// TIA Portal V17 export
// export: Created 2023-02-14T02:49:17.7051188Z, ExportSetting WithDefaults, DisplayName Totally Integrated Automation Portal, DisplayVersion V17, DisplayName TIA Portal Openness, DisplayVersion V17, DisplayName TIA Portal Teamcenter Gateway, DisplayVersion V17, DisplayName TIA Portal Version Control Interface, DisplayVersion V17, DisplayName SINAMICS Startdrive Advanced, DisplayVersion V17, DisplayName SINAMICS Startdrive G130, G150, S120, S150, SINAMICS MV, S210, DisplayVersion V17, DisplayName SINAMICS Startdrive G110M, G120, G120C, G120D, G120P, G115D, DisplayVersion V17, DisplayName STEP 7 Professional, DisplayVersion V17, DisplayName STEP 7 Safety, DisplayVersion V17, DisplayName WinCC Professional, DisplayVersion V17
FUNCTION "BlendingArea" : Void   // FC201, LAD
{ S7_Optimized_Access := 'TRUE' }
VERSION : 0.1
// stored: AutoNumber false, IsIECCheckEnabled false, SetENOAutomatically false, UDAEnableTagReadback false
   VAR_TEMP   // added for the SCL form of the ladder/FBD networks
      _w1 : Bool;
      _w2 : Bool;
   END_VAR
BEGIN

REGION Network 1: Analog
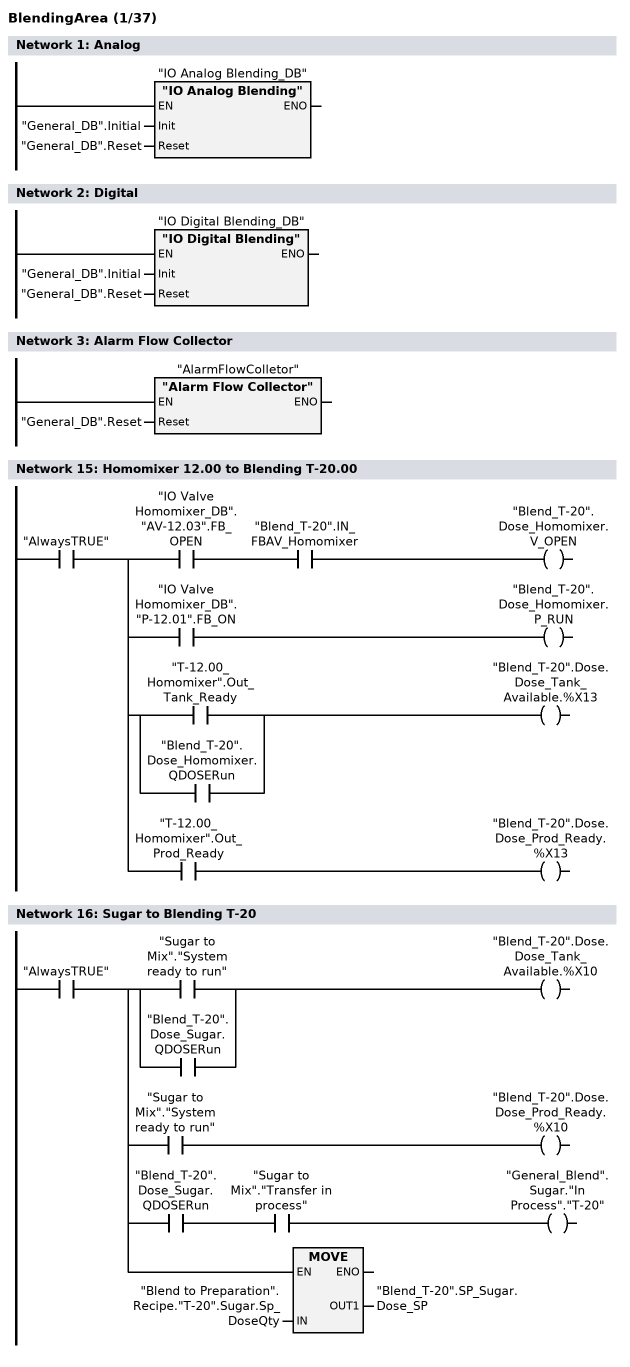
   RUNG wire#powerrail
      "IO Analog Blending_DB"(Init := "General_DB".Initial, Reset := "General_DB".Reset)
   END_RUNG
   // the same network as SCL:
   "IO Analog Blending_DB"(Init := "General_DB".Initial, Reset := "General_DB".Reset);   // "IO Analog Blending"
END_REGION

REGION Network 2: Digital
   RUNG wire#powerrail
      "IO Digital Blending_DB"(Init := "General_DB".Initial, Reset := "General_DB".Reset)
   END_RUNG
   // the same network as SCL:
   "IO Digital Blending_DB"(Init := "General_DB".Initial, Reset := "General_DB".Reset);   // "IO Digital Blending"
END_REGION

REGION Network 3: Alarm Flow Collector
   RUNG wire#powerrail
      "AlarmFlowColletor"(Reset := "General_DB".Reset)
   END_RUNG
   // the same network as SCL:
   "AlarmFlowColletor"(Reset := "General_DB".Reset);   // "Alarm Flow Collector"
END_REGION

NETWORK
TITLE = ChiliAwetan1 to Blending T-20
//Valve Open
      A     "Preparation to Blend"."T-02_ChiliAwetan_1".Valve_Open;
      A(;
      O(;
      A     "Blend_T-20".Dose.Dose_Header_Req.%X0;
      A     "Blend_T-20".IN_FBAV_Header1;
      );
      O(;
      A     "Blend_T-20".Dose.Dose_Header_Req.%X16;
      A     "Blend_T-20".IN_FBAV_Header2;
      );
      );
      =     "Blend_T-20".Dose_ChiliAwetan1.V_OPEN;
//Pump On
      O     "Preparation to Blend"."T-02_ChiliAwetan_1".Pump_Run;
      =     "Blend_T-20".Dose_ChiliAwetan1.P_RUN;
//Tank Available
      O     "Preparation to Blend"."T-02_ChiliAwetan_1".Tank_Available;
      O     "Blend_T-20".Dose_ChiliAwetan1.QDOSERun;
      =     "Blend_T-20".Dose.Dose_Tank_Available.%X0;
//Product Ready
      O     "Preparation to Blend"."T-02_ChiliAwetan_1".Product_Ready;
      =     "Blend_T-20".Dose.Dose_Prod_Ready.%X0;
//Level Tank
      L     "Preparation to Blend"."T-02_ChiliAwetan_1".Level;
      T     "Blend_T-20"."Dose_Level_%"."ChiliAwetan1%";


NETWORK
TITLE = ChiliAwetan2 to Blending T-20
//Valve Open
      A     "Preparation to Blend"."T-03_ChiliAwetan_2".Valve_Open;
      A(;
      O(;
      A     "Blend_T-20".Dose.Dose_Header_Req.%X1;
      A     "Blend_T-20".IN_FBAV_Header1;
      );
      O(;
      A     "Blend_T-20".Dose.Dose_Header_Req.%X17;
      A     "Blend_T-20".IN_FBAV_Header2;
      );
      );
      =     "Blend_T-20".Dose_ChiliAwetan2.V_OPEN;
//Pump On
      O     "Preparation to Blend"."T-03_ChiliAwetan_2".Pump_Run;
      =     "Blend_T-20".Dose_ChiliAwetan2.P_RUN;
//Tank Available
      O     "Preparation to Blend"."T-03_ChiliAwetan_2".Tank_Available;
      O     "Blend_T-20".Dose_ChiliAwetan2.QDOSERun;
      =     "Blend_T-20".Dose.Dose_Tank_Available.%X1;
//Product Ready
      O     "Preparation to Blend"."T-03_ChiliAwetan_2".Product_Ready;
      =     "Blend_T-20".Dose.Dose_Prod_Ready.%X1;
//Level Tank
      L     "Preparation to Blend"."T-03_ChiliAwetan_2".Level;
      T     "Blend_T-20"."Dose_Level_%"."ChiliAwetan2%";


NETWORK
TITLE = ChiliAwetan3 to Blending T-20
//Valve Open
      A     "Preparation to Blend"."T-04_ChiliAwetan_3".Valve_Open;
      A(;
      O(;
      A     "Blend_T-20".Dose.Dose_Header_Req.%X2;
      A     "Blend_T-20".IN_FBAV_Header1;
      );
      O(;
      A     "Blend_T-20".Dose.Dose_Header_Req.%X18;
      A     "Blend_T-20".IN_FBAV_Header2;
      );
      );
      =     "Blend_T-20".Dose_ChiliAwetan3.V_OPEN;
//Pump On
      O     "Preparation to Blend"."T-04_ChiliAwetan_3".Pump_Run;
      =     "Blend_T-20".Dose_ChiliAwetan3.P_RUN;
//Tank Available
      O     "Preparation to Blend"."T-04_ChiliAwetan_3".Tank_Available;
      O     "Blend_T-20".Dose_ChiliAwetan3.QDOSERun;
      =     "Blend_T-20".Dose.Dose_Tank_Available.%X2;
//Product Ready
      O     "Preparation to Blend"."T-04_ChiliAwetan_3".Product_Ready;
      =     "Blend_T-20".Dose.Dose_Prod_Ready.%X2;
//Level Tank
      L     "Preparation to Blend"."T-04_ChiliAwetan_3".Level;
      T     "Blend_T-20"."Dose_Level_%"."ChiliAwetan3%";


NETWORK
TITLE = Tomato to Blending T-20
//Valve Open
      A     "Preparation to Blend"."T-05_Tomato".Valve_Open;
      A(;
      O(;
      A     "Blend_T-20".Dose.Dose_Header_Req.%X3;
      A     "Blend_T-20".IN_FBAV_Header1;
      );
      O(;
      A     "Blend_T-20".Dose.Dose_Header_Req.%X19;
      A     "Blend_T-20".IN_FBAV_Header2;
      );
      );
      =     "Blend_T-20".Dose_Tomato.V_OPEN;
//Pump On
      O     "Preparation to Blend"."T-05_Tomato".Pump_Run;
      =     "Blend_T-20".Dose_Tomato.P_RUN;
//Tank Available
      O     "Preparation to Blend"."T-05_Tomato".Tank_Available;
      O     "Blend_T-20".Dose_Tomato.QDOSERun;
      =     "Blend_T-20".Dose.Dose_Tank_Available.%X3;
//Product Ready
      O     "Preparation to Blend"."T-05_Tomato".Product_Ready;
      =     "Blend_T-20".Dose.Dose_Prod_Ready.%X3;
//Level Tank
      L     "Preparation to Blend"."T-05_Tomato".Level;
      T     "Blend_T-20"."Dose_Level_%"."Tomato%";


NETWORK
TITLE = ChiliFresh1 to Blending T-20
//Valve Open
      A     "Preparation to Blend"."T-06_ChiliFresh_1".Valve_Open;
      A(;
      O(;
      A     "Blend_T-20".Dose.Dose_Header_Req.%X4;
      A     "Blend_T-20".IN_FBAV_Header1;
      );
      O(;
      A     "Blend_T-20".Dose.Dose_Header_Req.%X20;
      A     "Blend_T-20".IN_FBAV_Header2;
      );
      );
      =     "Blend_T-20".Dose_ChiliFresh1.V_OPEN;
//Pump On
      O     "Preparation to Blend"."T-06_ChiliFresh_1".Pump_Run;
      =     "Blend_T-20".Dose_ChiliFresh1.P_RUN;
//Tank Available
      O     "Preparation to Blend"."T-06_ChiliFresh_1".Tank_Available;
      O     "Blend_T-20".Dose_ChiliFresh1.QDOSERun;
      =     "Blend_T-20".Dose.Dose_Tank_Available.%X4;
//Product Ready
      O     "Preparation to Blend"."T-06_ChiliFresh_1".Product_Ready;
      =     "Blend_T-20".Dose.Dose_Prod_Ready.%X4;
//Level Tank
      L     "Preparation to Blend"."T-06_ChiliFresh_1".Level;
      T     "Blend_T-20"."Dose_Level_%"."ChiliFresh1%";


NETWORK
TITLE = ChiliFresh2 to Blending T-20
//Valve Open
      A     "Preparation to Blend"."T-07_ChiliFresh_2".Valve_Open;
      A(;
      O(;
      A     "Blend_T-20".Dose.Dose_Header_Req.%X5;
      A     "Blend_T-20".IN_FBAV_Header1;
      );
      O(;
      A     "Blend_T-20".Dose.Dose_Header_Req.%X21;
      A     "Blend_T-20".IN_FBAV_Header2;
      );
      );
      =     "Blend_T-20".Dose_ChiliFresh2.V_OPEN;
//Pump On
      O     "Preparation to Blend"."T-07_ChiliFresh_2".Pump_Run;
      =     "Blend_T-20".Dose_ChiliFresh2.P_RUN;
//Tank Available
      O     "Preparation to Blend"."T-07_ChiliFresh_2".Tank_Available;
      O     "Blend_T-20".Dose_ChiliFresh2.QDOSERun;
      =     "Blend_T-20".Dose.Dose_Tank_Available.%X5;
//Product Ready
      O     "Preparation to Blend"."T-07_ChiliFresh_2".Product_Ready;
      =     "Blend_T-20".Dose.Dose_Prod_Ready.%X5;
//Level Tank
      L     "Preparation to Blend"."T-07_ChiliFresh_2".Level;
      T     "Blend_T-20"."Dose_Level_%"."ChiliFresh2%";


NETWORK
TITLE = ChiliFresh3 to Blending T-20
//Valve Open
      A     "Preparation to Blend"."T-08_ChiliFresh_3".Valve_Open;
      A(;
      O(;
      A     "Blend_T-20".Dose.Dose_Header_Req.%X6;
      A     "Blend_T-20".IN_FBAV_Header1;
      );
      O(;
      A     "Blend_T-20".Dose.Dose_Header_Req.%X22;
      A     "Blend_T-20".IN_FBAV_Header2;
      );
      );
      =     "Blend_T-20".Dose_ChiliFresh3.V_OPEN;
//Pump On
      O     "Preparation to Blend"."T-08_ChiliFresh_3".Pump_Run;
      =     "Blend_T-20".Dose_ChiliFresh3.P_RUN;
//Tank Available
      O     "Preparation to Blend"."T-08_ChiliFresh_3".Tank_Available;
      O     "Blend_T-20".Dose_ChiliFresh3.QDOSERun;
      =     "Blend_T-20".Dose.Dose_Tank_Available.%X6;
//Product Ready
      O     "Preparation to Blend"."T-08_ChiliFresh_3".Product_Ready;
      =     "Blend_T-20".Dose.Dose_Prod_Ready.%X6;
//Level Tank
      L     "Preparation to Blend"."T-08_ChiliFresh_3".Level;
      T     "Blend_T-20"."Dose_Level_%"."ChiliFresh3%";


NETWORK
TITLE = Garlic to Blending T-20
//Valve Open
      A     "Preparation to Blend"."T-09_Garlic".Valve_Open;
      A(;
      O(;
      A     "Blend_T-20".Dose.Dose_Header_Req.%X7;
      A     "Blend_T-20".IN_FBAV_Header1;
      );
      O(;
      A     "Blend_T-20".Dose.Dose_Header_Req.%X23;
      A     "Blend_T-20".IN_FBAV_Header2;
      );
      );
      =     "Blend_T-20".Dose_Garlic.V_OPEN;
//Pump On
      O     "Preparation to Blend"."T-09_Garlic".Pump_Run;
      =     "Blend_T-20".Dose_Garlic.P_RUN;
//Tank Available
      O     "Preparation to Blend"."T-09_Garlic".Tank_Available;
      O     "Blend_T-20".Dose_Garlic.QDOSERun;
      =     "Blend_T-20".Dose.Dose_Tank_Available.%X7;
//Product Ready
      O     "Preparation to Blend"."T-09_Garlic".Product_Ready;
      =     "Blend_T-20".Dose.Dose_Prod_Ready.%X7;
//Level Tank
      L     "Preparation to Blend"."T-09_Garlic".Level;
      T     "Blend_T-20"."Dose_Level_%"."Garlic%";


NETWORK
TITLE = Vinegar to Blending T-20
//Valve Open
      A     "Preparation to Blend"."T-10_Vinegar".Valve_Open;
      A     "Blend_T-20".IN_FBAV_Vinegar;
      =     "Blend_T-20".Dose_Vinegar.V_OPEN;
//Pump On
      O     "Preparation to Blend"."T-10_Vinegar".Pump_Run;
      =     "Blend_T-20".Dose_Vinegar.P_RUN;
//Tank Available
      O     "Preparation to Blend"."T-10_Vinegar".Tank_Available;
      O     "Blend_T-20".Dose_Vinegar.QDOSERun;
      =     "Blend_T-20".Dose.Dose_Tank_Available.%X9;
//Product Ready
      O     "Preparation to Blend"."T-10_Vinegar".Product_Ready;
      =     "Blend_T-20".Dose.Dose_Prod_Ready.%X9;
//Level Tank
      L     "Preparation to Blend"."T-10_Vinegar".Level;
      T     "Blend_T-20"."Dose_Level_%"."Vinegar%";


NETWORK
TITLE = HW to Blending T-20
//Valve Open
      A     "Preparation to Blend"."T-51_HW".Valve_Open;
      A(;
      O(;
      A     "Blend_T-20".Dose.Dose_Header_Req.%X8;
      A     "Blend_T-20".IN_FBAV_Header1;
      );
      O(;
      A     "Blend_T-20".Dose.Dose_Header_Req.%X24;
      A     "Blend_T-20".IN_FBAV_Header2;
      );
      );
      =     "Blend_T-20".Dose_HW.V_OPEN;
//Pump On
      O     "Preparation to Blend"."T-51_HW".Pump_Run;
      =     "Blend_T-20".Dose_HW.P_RUN;
//Tank Available
      O     "Preparation to Blend"."T-51_HW".Tank_Available;
      O     "Blend_T-20".Dose_HW.QDOSERun;
      =     "Blend_T-20".Dose.Dose_Tank_Available.%X8;
//Product Ready
      O     "Preparation to Blend"."T-51_HW".Product_Ready;
      =     "Blend_T-20".Dose.Dose_Prod_Ready.%X8;
//Level Tank
// L     "Preparation to Blend"."T-01_HW".Level
// T     "Blend_T-20"."Dose_Level_%"."HW%"


REGION Network 15: Homomixer 12.00 to Blending T-20.00
   RUNG wire#powerrail
      Contact( "AlwaysTRUE" )
      wire#w1
      Contact( "IO Valve Homomixer_DB"."AV-12.03".FB_OPEN )
      Contact( "Blend_T-20".IN_FBAV_Homomixer )
      Coil( "Blend_T-20".Dose_Homomixer.V_OPEN )
   END_RUNG
   RUNG wire#w1
      Contact( "IO Valve Homomixer_DB"."P-12.01".FB_ON )
      Coil( "Blend_T-20".Dose_Homomixer.P_RUN )
   END_RUNG
   RUNG wire#w1
      Contact( "T-12.00_Homomixer".Out_Tank_Ready )
      wire#w2
      Coil( "Blend_T-20".Dose.Dose_Tank_Available.%X13 )
   END_RUNG
   RUNG wire#w1
      Contact( "Blend_T-20".Dose_Homomixer.QDOSERun )
   END_RUNG wire#w2
   RUNG wire#w1
      Contact( "T-12.00_Homomixer".Out_Prod_Ready )
      Coil( "Blend_T-20".Dose.Dose_Prod_Ready.%X13 )
   END_RUNG
   // the same network as SCL:
   "Blend_T-20".Dose_Homomixer.V_OPEN := "AlwaysTRUE" AND "IO Valve Homomixer_DB"."AV-12.03".FB_OPEN AND "Blend_T-20".IN_FBAV_Homomixer;
   "Blend_T-20".Dose_Homomixer.P_RUN := "AlwaysTRUE" AND "IO Valve Homomixer_DB"."P-12.01".FB_ON;
   "Blend_T-20".Dose.Dose_Tank_Available.%X13 := "AlwaysTRUE" AND ("T-12.00_Homomixer".Out_Tank_Ready OR "Blend_T-20".Dose_Homomixer.QDOSERun);
   "Blend_T-20".Dose.Dose_Prod_Ready.%X13 := "AlwaysTRUE" AND "T-12.00_Homomixer".Out_Prod_Ready;
END_REGION

REGION Network 16: Sugar to Blending T-20
   RUNG wire#powerrail
      Contact( "AlwaysTRUE" )
      wire#w1
      Contact( "Sugar to Mix"."System ready to run" )
      wire#w2
      Coil( "Blend_T-20".Dose.Dose_Tank_Available.%X10 )
   END_RUNG
   RUNG wire#w1
      Contact( "Blend_T-20".Dose_Sugar.QDOSERun )
   END_RUNG wire#w2
   RUNG wire#w1
      Contact( "Sugar to Mix"."System ready to run" )
      Coil( "Blend_T-20".Dose.Dose_Prod_Ready.%X10 )
   END_RUNG
   RUNG wire#w1
      Contact( "Blend_T-20".Dose_Sugar.QDOSERun )
      Contact( "Sugar to Mix"."Transfer in process" )
      Coil( "General_Blend".Sugar."In Process"."T-20" )
   END_RUNG
   RUNG wire#w1
      Move(in := "Blend to Preparation".Recipe."T-20".Sugar.Sp_DoseQty, out1 => "Blend_T-20".SP_Sugar.Dose_SP)
   END_RUNG
   // the same network as SCL:
   "Blend_T-20".Dose.Dose_Tank_Available.%X10 := "AlwaysTRUE" AND ("Sugar to Mix"."System ready to run" OR "Blend_T-20".Dose_Sugar.QDOSERun);
   "Blend_T-20".Dose.Dose_Prod_Ready.%X10 := "AlwaysTRUE" AND "Sugar to Mix"."System ready to run";
   "General_Blend".Sugar."In Process"."T-20" := "AlwaysTRUE" AND "Blend_T-20".Dose_Sugar.QDOSERun AND "Sugar to Mix"."Transfer in process";
   IF "AlwaysTRUE" THEN
       "Blend_T-20".SP_Sugar.Dose_SP := "Blend to Preparation".Recipe."T-20".Sugar.Sp_DoseQty;
   END_IF;
END_REGION

REGION Network 17: Salt to Blending T-20
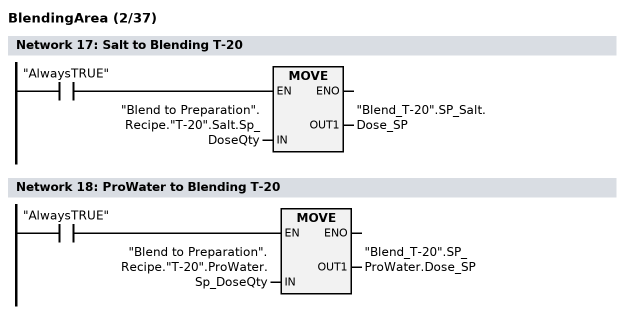
   RUNG wire#powerrail
      Contact( "AlwaysTRUE" )
      Move(in := "Blend to Preparation".Recipe."T-20".Salt.Sp_DoseQty, out1 => "Blend_T-20".SP_Salt.Dose_SP)
   END_RUNG
   // the same network as SCL:
   IF "AlwaysTRUE" THEN
       "Blend_T-20".SP_Salt.Dose_SP := "Blend to Preparation".Recipe."T-20".Salt.Sp_DoseQty;
   END_IF;
END_REGION

REGION Network 18: ProWater to Blending T-20
   RUNG wire#powerrail
      Contact( "AlwaysTRUE" )
      Move(in := "Blend to Preparation".Recipe."T-20".ProWater.Sp_DoseQty, out1 => "Blend_T-20".SP_ProWater.Dose_SP)
   END_RUNG
   // the same network as SCL:
   IF "AlwaysTRUE" THEN
       "Blend_T-20".SP_ProWater.Dose_SP := "Blend to Preparation".Recipe."T-20".ProWater.Sp_DoseQty;
   END_IF;
END_REGION

REGION Network 19: Blending T-20
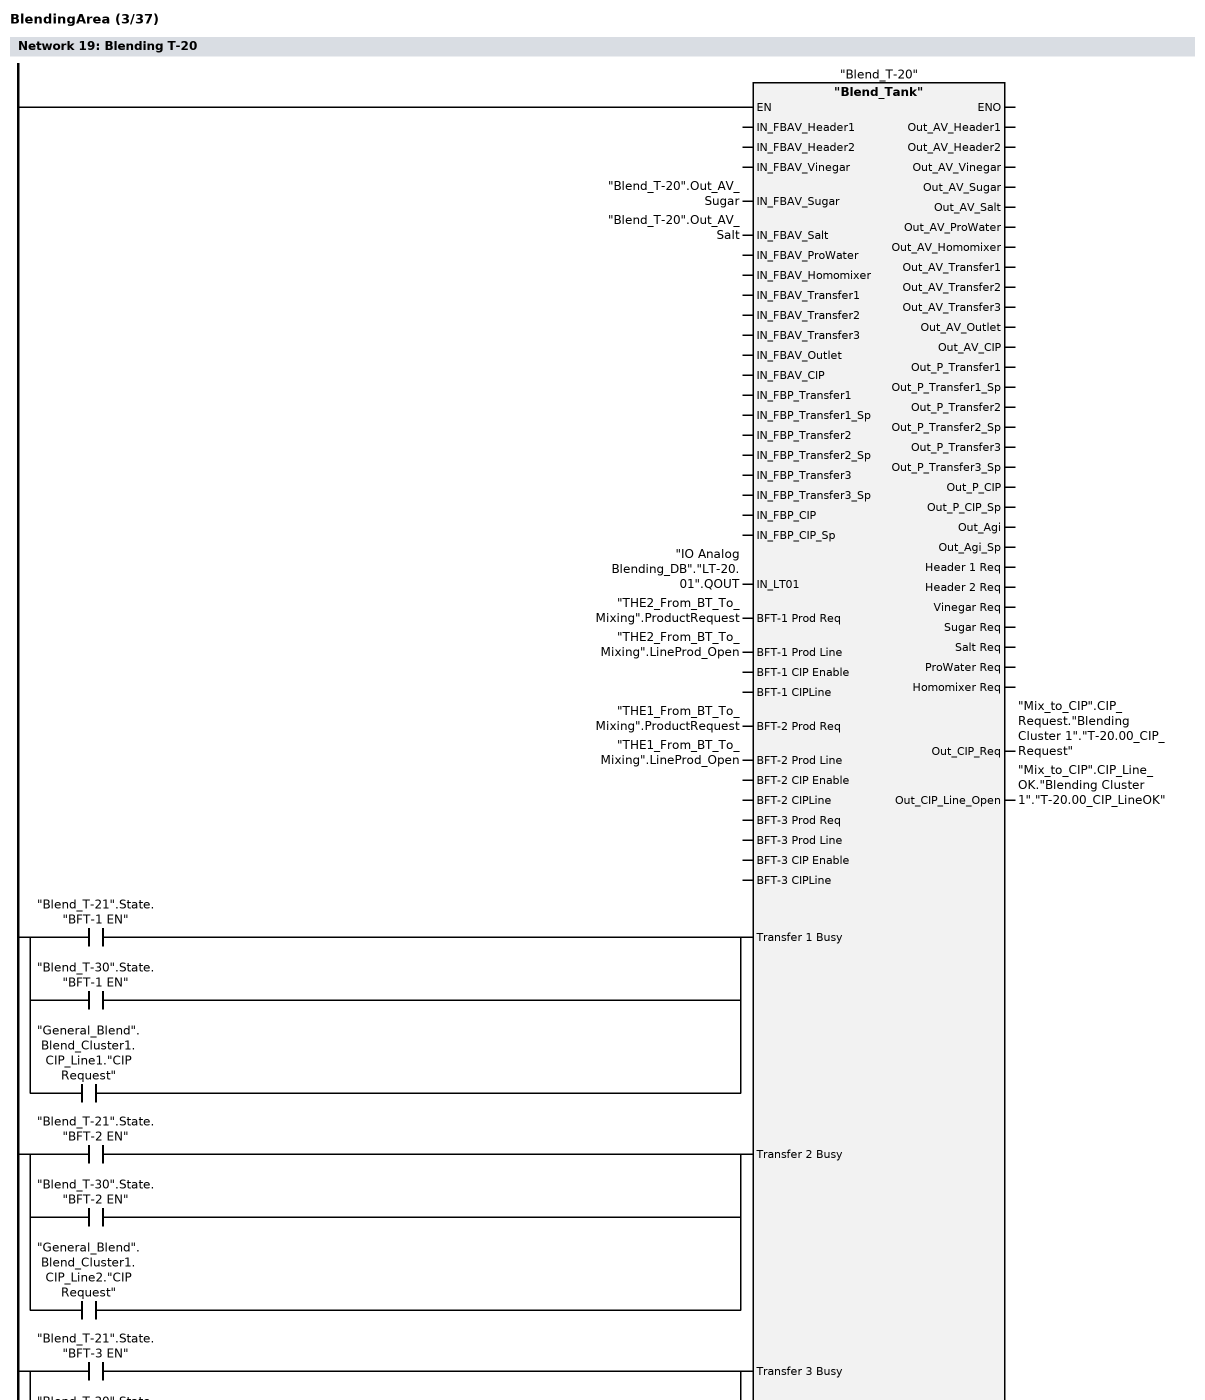
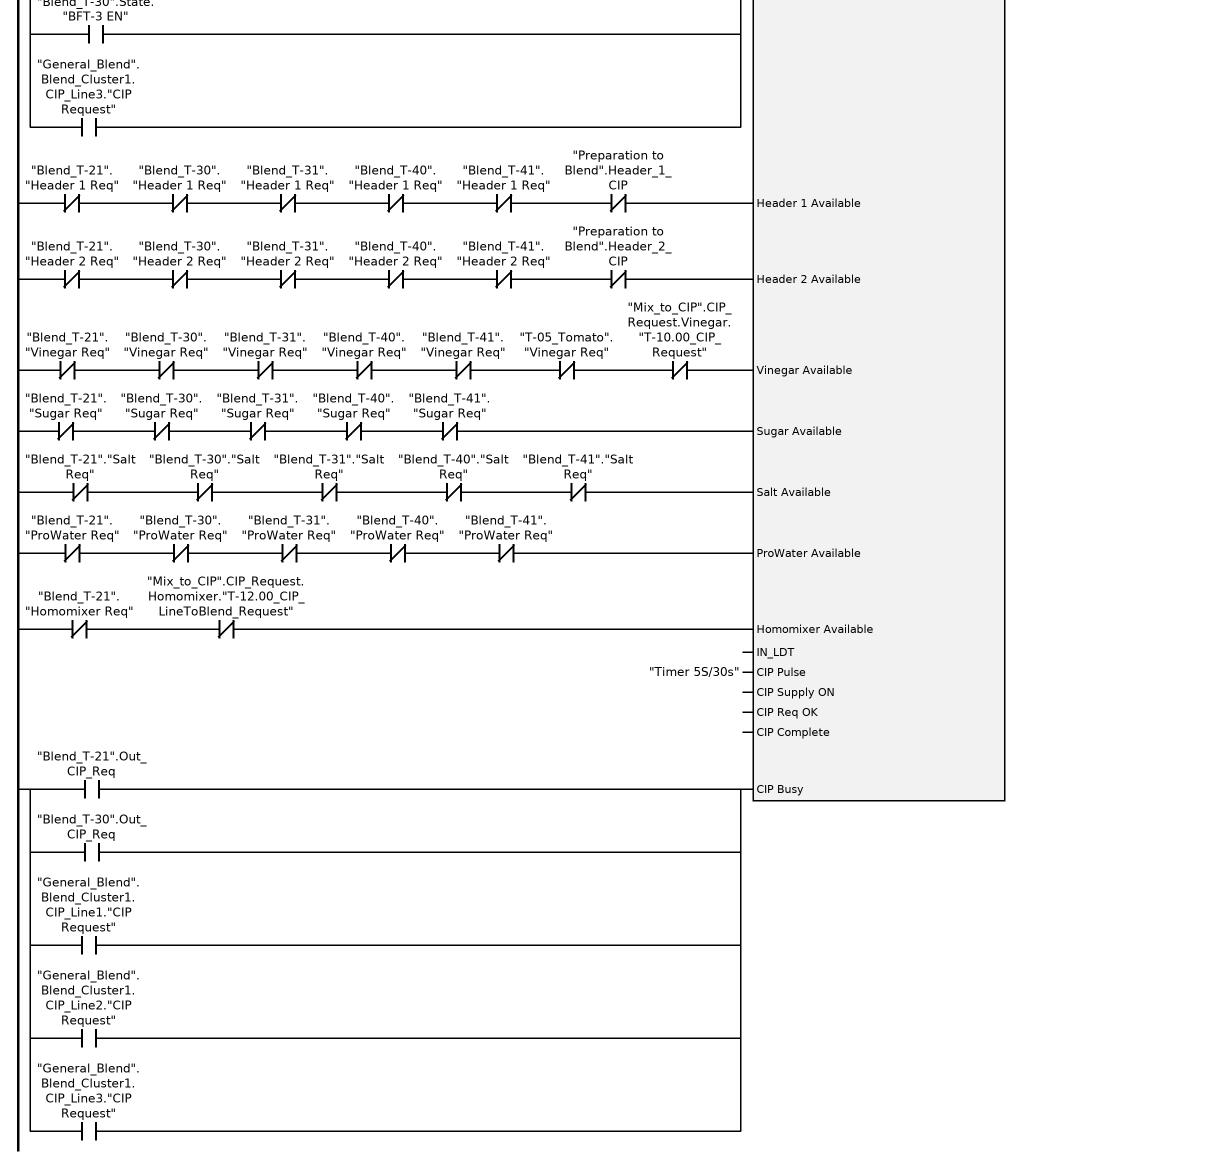
   RUNG wire#powerrail
      "Blend_T-20"("Transfer 1 Busy" := wire#w1, "Transfer 2 Busy" := wire#w2, "Transfer 3 Busy" := wire#w3, "Header 1 Available" := wire#w4, "Header 2 Available" := wire#w5, "Vinegar Available" := wire#w6, "Sugar Available" := wire#w7, "Salt Available" := wire#w8, "ProWater Available" := wire#w9, "Homomixer Available" := wire#w10, "CIP Busy" := wire#w11, IN_FBAV_Header1 :=, IN_FBAV_Header2 :=, IN_FBAV_Vinegar :=, IN_FBAV_Sugar := "Blend_T-20".Out_AV_Sugar, IN_FBAV_Salt := "Blend_T-20".Out_AV_Salt, IN_FBAV_ProWater :=, IN_FBAV_Homomixer :=, IN_FBAV_Transfer1 :=, IN_FBAV_Transfer2 :=, IN_FBAV_Transfer3 :=, IN_FBAV_Outlet :=, IN_FBAV_CIP :=, IN_FBP_Transfer1 :=, IN_FBP_Transfer1_Sp :=, IN_FBP_Transfer2 :=, IN_FBP_Transfer2_Sp :=, IN_FBP_Transfer3 :=, IN_FBP_Transfer3_Sp :=, IN_FBP_CIP :=, IN_FBP_CIP_Sp :=, IN_LT01 := "IO Analog Blending_DB"."LT-20.01".QOUT, "BFT-1 Prod Req" := "THE2_From_BT_To_Mixing".ProductRequest, "BFT-1 Prod Line" := "THE2_From_BT_To_Mixing".LineProd_Open, "BFT-1 CIP Enable" :=, "BFT-1 CIPLine" :=, "BFT-2 Prod Req" := "THE1_From_BT_To_Mixing".ProductRequest, "BFT-2 Prod Line" := "THE1_From_BT_To_Mixing".LineProd_Open, "BFT-2 CIP Enable" :=, "BFT-2 CIPLine" :=, "BFT-3 Prod Req" :=, "BFT-3 Prod Line" :=, "BFT-3 CIP Enable" :=, "BFT-3 CIPLine" :=, IN_LDT :=, "CIP Pulse" := "Timer 5S/30s", "CIP Supply ON" :=, "CIP Req OK" :=, "CIP Complete" :=, Out_AV_Header1 =>, Out_AV_Header2 =>, Out_AV_Vinegar =>, Out_AV_Sugar =>, Out_AV_Salt =>, Out_AV_ProWater =>, Out_AV_Homomixer =>, Out_AV_Transfer1 =>, Out_AV_Transfer2 =>, Out_AV_Transfer3 =>, Out_AV_Outlet =>, Out_AV_CIP =>, Out_P_Transfer1 =>, Out_P_Transfer1_Sp =>, Out_P_Transfer2 =>, Out_P_Transfer2_Sp =>, Out_P_Transfer3 =>, Out_P_Transfer3_Sp =>, Out_P_CIP =>, Out_P_CIP_Sp =>, Out_Agi =>, Out_Agi_Sp =>, "Header 1 Req" =>, "Header 2 Req" =>, "Vinegar Req" =>, "Sugar Req" =>, "Salt Req" =>, "ProWater Req" =>, "Homomixer Req" =>, Out_CIP_Req => "Mix_to_CIP".CIP_Request."Blending Cluster 1"."T-20.00_CIP_Request", Out_CIP_Line_Open => "Mix_to_CIP".CIP_Line_OK."Blending Cluster 1"."T-20.00_CIP_LineOK")
   END_RUNG
   RUNG wire#powerrail
      Contact( "Blend_T-21".State."BFT-1 EN" )
   END_RUNG wire#w1
   RUNG wire#powerrail
      Contact( "Blend_T-30".State."BFT-1 EN" )
   END_RUNG wire#w1
   RUNG wire#powerrail
      Contact( "General_Blend".Blend_Cluster1.CIP_Line1."CIP Request" )
   END_RUNG wire#w1
   RUNG wire#powerrail
      Contact( "Blend_T-21".State."BFT-2 EN" )
   END_RUNG wire#w2
   RUNG wire#powerrail
      Contact( "Blend_T-30".State."BFT-2 EN" )
   END_RUNG wire#w2
   RUNG wire#powerrail
      Contact( "General_Blend".Blend_Cluster1.CIP_Line2."CIP Request" )
   END_RUNG wire#w2
   RUNG wire#powerrail
      Contact( "Blend_T-21".State."BFT-3 EN" )
   END_RUNG wire#w3
   RUNG wire#powerrail
      Contact( "Blend_T-30".State."BFT-3 EN" )
   END_RUNG wire#w3
   RUNG wire#powerrail
      Contact( "General_Blend".Blend_Cluster1.CIP_Line3."CIP Request" )
   END_RUNG wire#w3
   RUNG wire#powerrail
      I_Contact( "Blend_T-21"."Header 1 Req" )
      I_Contact( "Blend_T-30"."Header 1 Req" )
      I_Contact( "Blend_T-31"."Header 1 Req" )
      I_Contact( "Blend_T-40"."Header 1 Req" )
      I_Contact( "Blend_T-41"."Header 1 Req" )
      I_Contact( "Preparation to Blend".Header_1_CIP )
   END_RUNG wire#w4
   RUNG wire#powerrail
      I_Contact( "Blend_T-21"."Header 2 Req" )
      I_Contact( "Blend_T-30"."Header 2 Req" )
      I_Contact( "Blend_T-31"."Header 2 Req" )
      I_Contact( "Blend_T-40"."Header 2 Req" )
      I_Contact( "Blend_T-41"."Header 2 Req" )
      I_Contact( "Preparation to Blend".Header_2_CIP )
   END_RUNG wire#w5
   RUNG wire#powerrail
      I_Contact( "Blend_T-21"."Vinegar Req" )
      I_Contact( "Blend_T-30"."Vinegar Req" )
      I_Contact( "Blend_T-31"."Vinegar Req" )
      I_Contact( "Blend_T-40"."Vinegar Req" )
      I_Contact( "Blend_T-41"."Vinegar Req" )
      I_Contact( "T-05_Tomato"."Vinegar Req" )
      I_Contact( "Mix_to_CIP".CIP_Request.Vinegar."T-10.00_CIP_Request" )
   END_RUNG wire#w6
   RUNG wire#powerrail
      I_Contact( "Blend_T-21"."Sugar Req" )
      I_Contact( "Blend_T-30"."Sugar Req" )
      I_Contact( "Blend_T-31"."Sugar Req" )
      I_Contact( "Blend_T-40"."Sugar Req" )
      I_Contact( "Blend_T-41"."Sugar Req" )
   END_RUNG wire#w7
   RUNG wire#powerrail
      I_Contact( "Blend_T-21"."Salt Req" )
      I_Contact( "Blend_T-30"."Salt Req" )
      I_Contact( "Blend_T-31"."Salt Req" )
      I_Contact( "Blend_T-40"."Salt Req" )
      I_Contact( "Blend_T-41"."Salt Req" )
   END_RUNG wire#w8
   RUNG wire#powerrail
      I_Contact( "Blend_T-21"."ProWater Req" )
      I_Contact( "Blend_T-30"."ProWater Req" )
      I_Contact( "Blend_T-31"."ProWater Req" )
      I_Contact( "Blend_T-40"."ProWater Req" )
      I_Contact( "Blend_T-41"."ProWater Req" )
   END_RUNG wire#w9
   RUNG wire#powerrail
      I_Contact( "Blend_T-21"."Homomixer Req" )
      I_Contact( "Mix_to_CIP".CIP_Request.Homomixer."T-12.00_CIP_LineToBlend_Request" )
   END_RUNG wire#w10
   RUNG wire#powerrail
      Contact( "Blend_T-21".Out_CIP_Req )
   END_RUNG wire#w11
   RUNG wire#powerrail
      Contact( "Blend_T-30".Out_CIP_Req )
   END_RUNG wire#w11
   RUNG wire#powerrail
      Contact( "General_Blend".Blend_Cluster1.CIP_Line1."CIP Request" )
   END_RUNG wire#w11
   RUNG wire#powerrail
      Contact( "General_Blend".Blend_Cluster1.CIP_Line2."CIP Request" )
   END_RUNG wire#w11
   RUNG wire#powerrail
      Contact( "General_Blend".Blend_Cluster1.CIP_Line3."CIP Request" )
   END_RUNG wire#w11
   // the same network as SCL:
   "Blend_T-20"(IN_FBAV_Sugar := "Blend_T-20".Out_AV_Sugar,   // "Blend_Tank"
                IN_FBAV_Salt := "Blend_T-20".Out_AV_Salt,
                IN_LT01 := "IO Analog Blending_DB"."LT-20.01".QOUT,
                "BFT-1 Prod Req" := "THE2_From_BT_To_Mixing".ProductRequest,
                "BFT-1 Prod Line" := "THE2_From_BT_To_Mixing".LineProd_Open,
                "BFT-2 Prod Req" := "THE1_From_BT_To_Mixing".ProductRequest,
                "BFT-2 Prod Line" := "THE1_From_BT_To_Mixing".LineProd_Open,
                "Transfer 1 Busy" := "Blend_T-21".State."BFT-1 EN" OR "Blend_T-30".State."BFT-1 EN" OR "General_Blend".Blend_Cluster1.CIP_Line1."CIP Request",
                "Transfer 2 Busy" := "Blend_T-21".State."BFT-2 EN" OR "Blend_T-30".State."BFT-2 EN" OR "General_Blend".Blend_Cluster1.CIP_Line2."CIP Request",
                "Transfer 3 Busy" := "Blend_T-21".State."BFT-3 EN" OR "Blend_T-30".State."BFT-3 EN" OR "General_Blend".Blend_Cluster1.CIP_Line3."CIP Request",
                "Header 1 Available" := NOT "Blend_T-21"."Header 1 Req" AND NOT "Blend_T-30"."Header 1 Req" AND NOT "Blend_T-31"."Header 1 Req" AND NOT "Blend_T-40"."Header 1 Req" AND NOT "Blend_T-41"."Header 1 Req" AND NOT "Preparation to Blend".Header_1_CIP,
                "Header 2 Available" := NOT "Blend_T-21"."Header 2 Req" AND NOT "Blend_T-30"."Header 2 Req" AND NOT "Blend_T-31"."Header 2 Req" AND NOT "Blend_T-40"."Header 2 Req" AND NOT "Blend_T-41"."Header 2 Req" AND NOT "Preparation to Blend".Header_2_CIP,
                "Vinegar Available" := NOT "Blend_T-21"."Vinegar Req" AND NOT "Blend_T-30"."Vinegar Req" AND NOT "Blend_T-31"."Vinegar Req" AND NOT "Blend_T-40"."Vinegar Req" AND NOT "Blend_T-41"."Vinegar Req" AND NOT "T-05_Tomato"."Vinegar Req" AND NOT "Mix_to_CIP".CIP_Request.Vinegar."T-10.00_CIP_Request",
                "Sugar Available" := NOT "Blend_T-21"."Sugar Req" AND NOT "Blend_T-30"."Sugar Req" AND NOT "Blend_T-31"."Sugar Req" AND NOT "Blend_T-40"."Sugar Req" AND NOT "Blend_T-41"."Sugar Req",
                "Salt Available" := NOT "Blend_T-21"."Salt Req" AND NOT "Blend_T-30"."Salt Req" AND NOT "Blend_T-31"."Salt Req" AND NOT "Blend_T-40"."Salt Req" AND NOT "Blend_T-41"."Salt Req",
                "ProWater Available" := NOT "Blend_T-21"."ProWater Req" AND NOT "Blend_T-30"."ProWater Req" AND NOT "Blend_T-31"."ProWater Req" AND NOT "Blend_T-40"."ProWater Req" AND NOT "Blend_T-41"."ProWater Req",
                "Homomixer Available" := NOT "Blend_T-21"."Homomixer Req" AND NOT "Mix_to_CIP".CIP_Request.Homomixer."T-12.00_CIP_LineToBlend_Request",
                "CIP Pulse" := "Timer 5S/30s",
                "CIP Busy" := "Blend_T-21".Out_CIP_Req OR "Blend_T-30".Out_CIP_Req OR "General_Blend".Blend_Cluster1.CIP_Line1."CIP Request" OR "General_Blend".Blend_Cluster1.CIP_Line2."CIP Request" OR "General_Blend".Blend_Cluster1.CIP_Line3."CIP Request",
                Out_CIP_Req => "Mix_to_CIP".CIP_Request."Blending Cluster 1"."T-20.00_CIP_Request",
                Out_CIP_Line_Open => "Mix_to_CIP".CIP_Line_OK."Blending Cluster 1"."T-20.00_CIP_LineOK");
END_REGION

REGION Network 20: Blending T-20 Feedback Valve
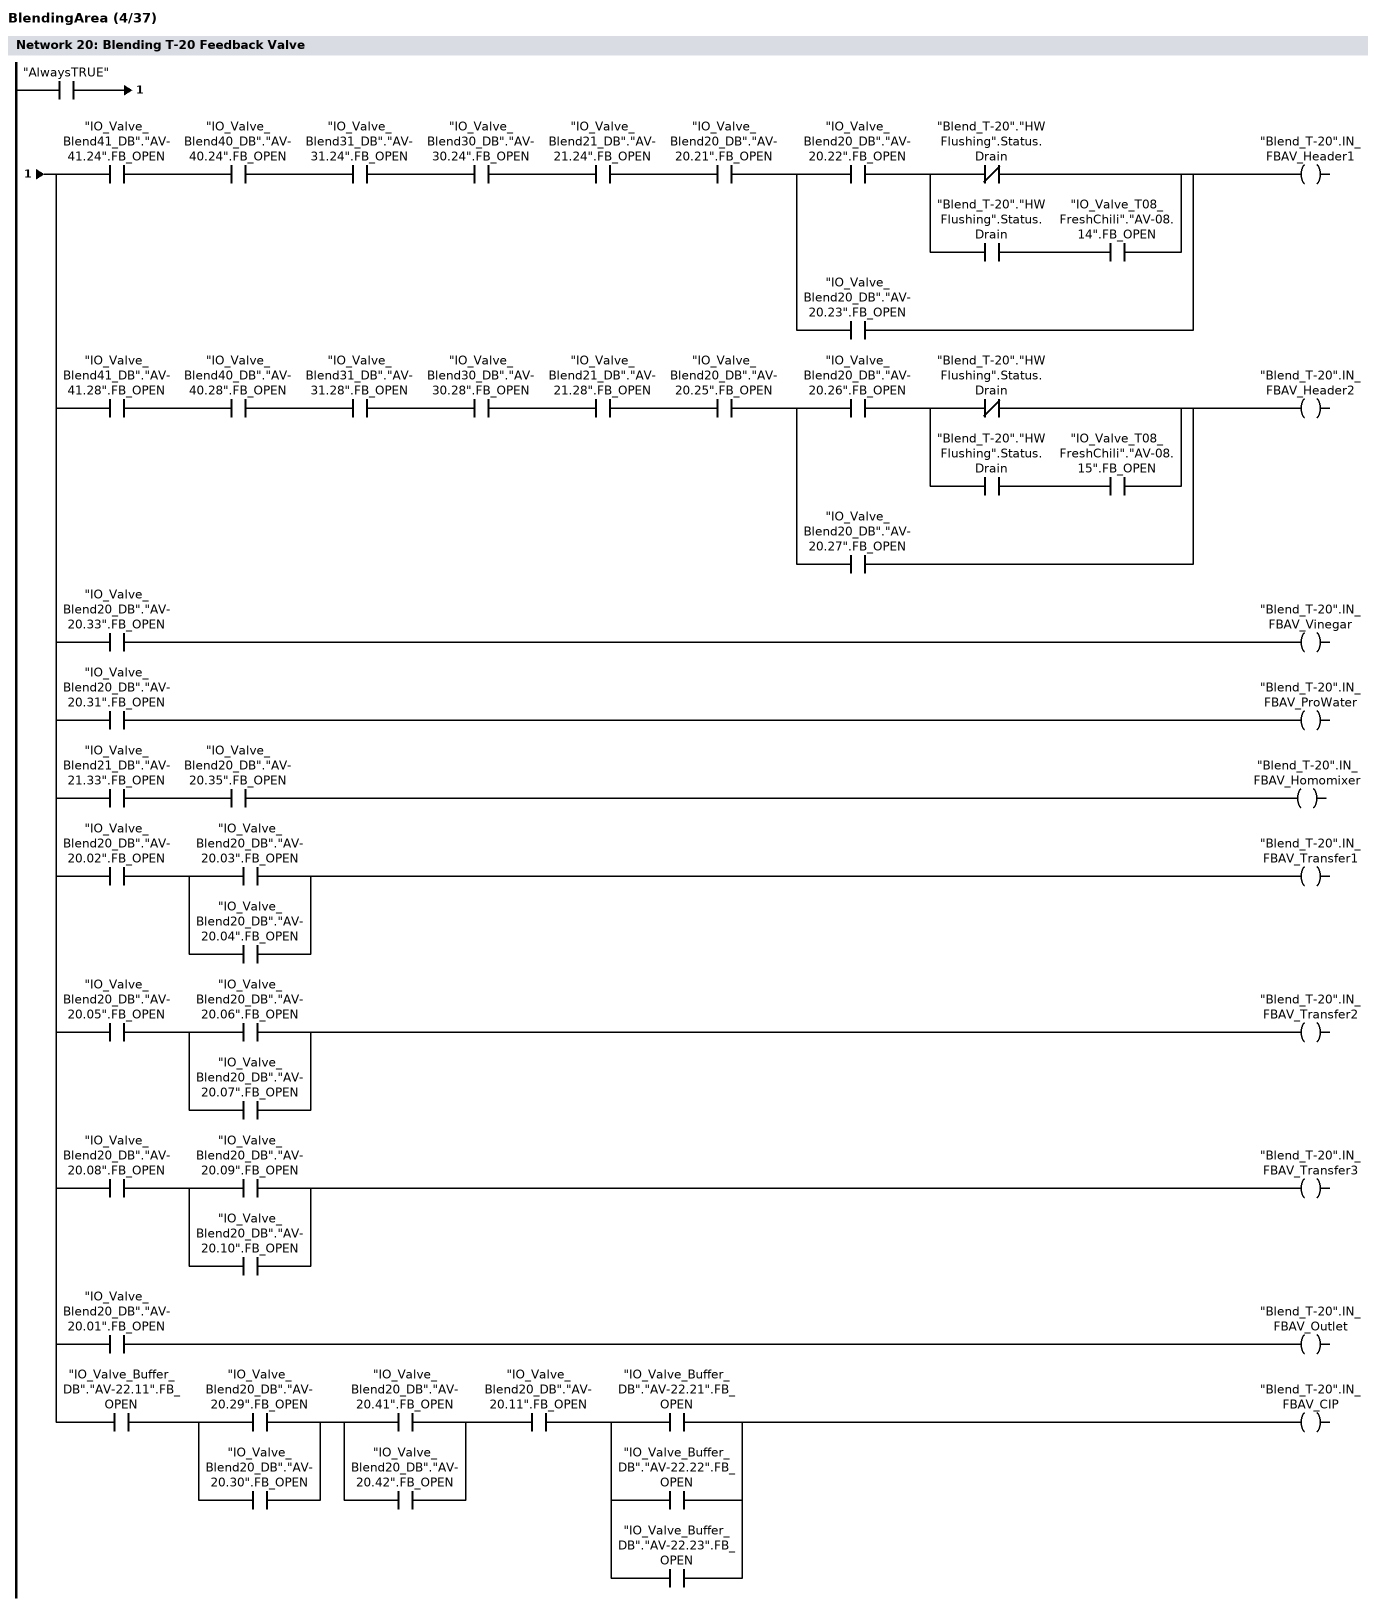
   RUNG wire#powerrail
      Contact( "AlwaysTRUE" )
      wire#w1
      Contact( "IO_Valve_Blend41_DB"."AV-41.24".FB_OPEN )
      Contact( "IO_Valve_Blend40_DB"."AV-40.24".FB_OPEN )
      Contact( "IO_Valve_Blend31_DB"."AV-31.24".FB_OPEN )
      Contact( "IO_Valve_Blend30_DB"."AV-30.24".FB_OPEN )
      Contact( "IO_Valve_Blend21_DB"."AV-21.24".FB_OPEN )
      Contact( "IO_Valve_Blend20_DB"."AV-20.21".FB_OPEN )
      wire#w2
      Contact( "IO_Valve_Blend20_DB"."AV-20.22".FB_OPEN )
      wire#w3
      I_Contact( "Blend_T-20"."HW Flushing".Status.Drain )
      wire#w4
      Coil( "Blend_T-20".IN_FBAV_Header1 )
   END_RUNG
   RUNG wire#w3
      Contact( "Blend_T-20"."HW Flushing".Status.Drain )
      Contact( "IO_Valve_T08_FreshChili"."AV-08.14".FB_OPEN )
   END_RUNG wire#w4
   RUNG wire#w2
      Contact( "IO_Valve_Blend20_DB"."AV-20.23".FB_OPEN )
   END_RUNG wire#w4
   RUNG wire#w1
      Contact( "IO_Valve_Blend41_DB"."AV-41.28".FB_OPEN )
      Contact( "IO_Valve_Blend40_DB"."AV-40.28".FB_OPEN )
      Contact( "IO_Valve_Blend31_DB"."AV-31.28".FB_OPEN )
      Contact( "IO_Valve_Blend30_DB"."AV-30.28".FB_OPEN )
      Contact( "IO_Valve_Blend21_DB"."AV-21.28".FB_OPEN )
      Contact( "IO_Valve_Blend20_DB"."AV-20.25".FB_OPEN )
      wire#w5
      Contact( "IO_Valve_Blend20_DB"."AV-20.26".FB_OPEN )
      wire#w6
      I_Contact( "Blend_T-20"."HW Flushing".Status.Drain )
      wire#w7
      Coil( "Blend_T-20".IN_FBAV_Header2 )
   END_RUNG
   RUNG wire#w6
      Contact( "Blend_T-20"."HW Flushing".Status.Drain )
      Contact( "IO_Valve_T08_FreshChili"."AV-08.15".FB_OPEN )
   END_RUNG wire#w7
   RUNG wire#w5
      Contact( "IO_Valve_Blend20_DB"."AV-20.27".FB_OPEN )
   END_RUNG wire#w7
   RUNG wire#w1
      Contact( "IO_Valve_Blend20_DB"."AV-20.33".FB_OPEN )
      Coil( "Blend_T-20".IN_FBAV_Vinegar )
   END_RUNG
   RUNG wire#w1
      Contact( "IO_Valve_Blend20_DB"."AV-20.31".FB_OPEN )
      Coil( "Blend_T-20".IN_FBAV_ProWater )
   END_RUNG
   RUNG wire#w1
      Contact( "IO_Valve_Blend21_DB"."AV-21.33".FB_OPEN )
      Contact( "IO_Valve_Blend20_DB"."AV-20.35".FB_OPEN )
      Coil( "Blend_T-20".IN_FBAV_Homomixer )
   END_RUNG
   RUNG wire#w1
      Contact( "IO_Valve_Blend20_DB"."AV-20.02".FB_OPEN )
      wire#w8
      Contact( "IO_Valve_Blend20_DB"."AV-20.03".FB_OPEN )
      wire#w9
      Coil( "Blend_T-20".IN_FBAV_Transfer1 )
   END_RUNG
   RUNG wire#w8
      Contact( "IO_Valve_Blend20_DB"."AV-20.04".FB_OPEN )
   END_RUNG wire#w9
   RUNG wire#w1
      Contact( "IO_Valve_Blend20_DB"."AV-20.05".FB_OPEN )
      wire#w10
      Contact( "IO_Valve_Blend20_DB"."AV-20.06".FB_OPEN )
      wire#w11
      Coil( "Blend_T-20".IN_FBAV_Transfer2 )
   END_RUNG
   RUNG wire#w10
      Contact( "IO_Valve_Blend20_DB"."AV-20.07".FB_OPEN )
   END_RUNG wire#w11
   RUNG wire#w1
      Contact( "IO_Valve_Blend20_DB"."AV-20.08".FB_OPEN )
      wire#w12
      Contact( "IO_Valve_Blend20_DB"."AV-20.09".FB_OPEN )
      wire#w13
      Coil( "Blend_T-20".IN_FBAV_Transfer3 )
   END_RUNG
   RUNG wire#w12
      Contact( "IO_Valve_Blend20_DB"."AV-20.10".FB_OPEN )
   END_RUNG wire#w13
   RUNG wire#w1
      Contact( "IO_Valve_Blend20_DB"."AV-20.01".FB_OPEN )
      Coil( "Blend_T-20".IN_FBAV_Outlet )
   END_RUNG
   RUNG wire#w1
      Contact( "IO_Valve_Buffer_DB"."AV-22.11".FB_OPEN )
      wire#w14
      Contact( "IO_Valve_Blend20_DB"."AV-20.29".FB_OPEN )
      wire#w15
      Contact( "IO_Valve_Blend20_DB"."AV-20.41".FB_OPEN )
      wire#w16
      Contact( "IO_Valve_Blend20_DB"."AV-20.11".FB_OPEN )
      wire#w17
      Contact( "IO_Valve_Buffer_DB"."AV-22.21".FB_OPEN )
      wire#w18
      Coil( "Blend_T-20".IN_FBAV_CIP )
   END_RUNG
   RUNG wire#w14
      Contact( "IO_Valve_Blend20_DB"."AV-20.30".FB_OPEN )
   END_RUNG wire#w15
   RUNG wire#w15
      Contact( "IO_Valve_Blend20_DB"."AV-20.42".FB_OPEN )
   END_RUNG wire#w16
   RUNG wire#w17
      Contact( "IO_Valve_Buffer_DB"."AV-22.22".FB_OPEN )
   END_RUNG wire#w18
   RUNG wire#w17
      Contact( "IO_Valve_Buffer_DB"."AV-22.23".FB_OPEN )
   END_RUNG wire#w18
   // the same network as SCL:
   "Blend_T-20".IN_FBAV_Header1 := "AlwaysTRUE" AND "IO_Valve_Blend41_DB"."AV-41.24".FB_OPEN AND "IO_Valve_Blend40_DB"."AV-40.24".FB_OPEN AND "IO_Valve_Blend31_DB"."AV-31.24".FB_OPEN AND "IO_Valve_Blend30_DB"."AV-30.24".FB_OPEN AND "IO_Valve_Blend21_DB"."AV-21.24".FB_OPEN AND "IO_Valve_Blend20_DB"."AV-20.21".FB_OPEN AND (("IO_Valve_Blend20_DB"."AV-20.22".FB_OPEN AND (NOT "Blend_T-20"."HW Flushing".Status.Drain OR ("Blend_T-20"."HW Flushing".Status.Drain AND "IO_Valve_T08_FreshChili"."AV-08.14".FB_OPEN))) OR "IO_Valve_Blend20_DB"."AV-20.23".FB_OPEN);
   "Blend_T-20".IN_FBAV_Header2 := "AlwaysTRUE" AND "IO_Valve_Blend41_DB"."AV-41.28".FB_OPEN AND "IO_Valve_Blend40_DB"."AV-40.28".FB_OPEN AND "IO_Valve_Blend31_DB"."AV-31.28".FB_OPEN AND "IO_Valve_Blend30_DB"."AV-30.28".FB_OPEN AND "IO_Valve_Blend21_DB"."AV-21.28".FB_OPEN AND "IO_Valve_Blend20_DB"."AV-20.25".FB_OPEN AND (("IO_Valve_Blend20_DB"."AV-20.26".FB_OPEN AND (NOT "Blend_T-20"."HW Flushing".Status.Drain OR ("Blend_T-20"."HW Flushing".Status.Drain AND "IO_Valve_T08_FreshChili"."AV-08.15".FB_OPEN))) OR "IO_Valve_Blend20_DB"."AV-20.27".FB_OPEN);
   "Blend_T-20".IN_FBAV_Vinegar := "AlwaysTRUE" AND "IO_Valve_Blend20_DB"."AV-20.33".FB_OPEN;
   "Blend_T-20".IN_FBAV_ProWater := "AlwaysTRUE" AND "IO_Valve_Blend20_DB"."AV-20.31".FB_OPEN;
   "Blend_T-20".IN_FBAV_Homomixer := "AlwaysTRUE" AND "IO_Valve_Blend21_DB"."AV-21.33".FB_OPEN AND "IO_Valve_Blend20_DB"."AV-20.35".FB_OPEN;
   "Blend_T-20".IN_FBAV_Transfer1 := "AlwaysTRUE" AND "IO_Valve_Blend20_DB"."AV-20.02".FB_OPEN AND ("IO_Valve_Blend20_DB"."AV-20.03".FB_OPEN OR "IO_Valve_Blend20_DB"."AV-20.04".FB_OPEN);
   "Blend_T-20".IN_FBAV_Transfer2 := "AlwaysTRUE" AND "IO_Valve_Blend20_DB"."AV-20.05".FB_OPEN AND ("IO_Valve_Blend20_DB"."AV-20.06".FB_OPEN OR "IO_Valve_Blend20_DB"."AV-20.07".FB_OPEN);
   "Blend_T-20".IN_FBAV_Transfer3 := "AlwaysTRUE" AND "IO_Valve_Blend20_DB"."AV-20.08".FB_OPEN AND ("IO_Valve_Blend20_DB"."AV-20.09".FB_OPEN OR "IO_Valve_Blend20_DB"."AV-20.10".FB_OPEN);
   "Blend_T-20".IN_FBAV_Outlet := "AlwaysTRUE" AND "IO_Valve_Blend20_DB"."AV-20.01".FB_OPEN;
   "Blend_T-20".IN_FBAV_CIP := "AlwaysTRUE" AND "IO_Valve_Buffer_DB"."AV-22.11".FB_OPEN AND ("IO_Valve_Blend20_DB"."AV-20.29".FB_OPEN OR "IO_Valve_Blend20_DB"."AV-20.30".FB_OPEN) AND ("IO_Valve_Blend20_DB"."AV-20.41".FB_OPEN OR "IO_Valve_Blend20_DB"."AV-20.42".FB_OPEN) AND "IO_Valve_Blend20_DB"."AV-20.11".FB_OPEN AND ("IO_Valve_Buffer_DB"."AV-22.21".FB_OPEN OR "IO_Valve_Buffer_DB"."AV-22.22".FB_OPEN OR "IO_Valve_Buffer_DB"."AV-22.23".FB_OPEN);
END_REGION

REGION Network 21: Blending T-20 Feedback Pump
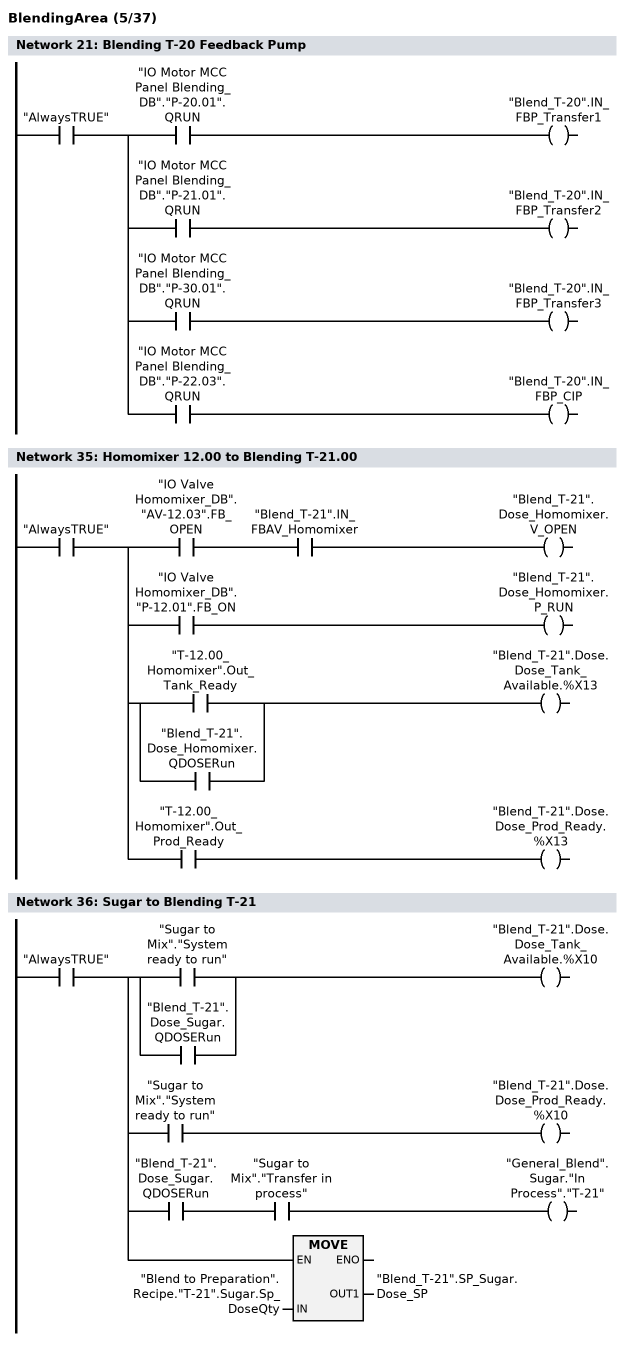
   RUNG wire#powerrail
      Contact( "AlwaysTRUE" )
      wire#w1
      Contact( "IO Motor MCC Panel Blending_DB"."P-20.01".QRUN )
      Coil( "Blend_T-20".IN_FBP_Transfer1 )
   END_RUNG
   RUNG wire#w1
      Contact( "IO Motor MCC Panel Blending_DB"."P-21.01".QRUN )
      Coil( "Blend_T-20".IN_FBP_Transfer2 )
   END_RUNG
   RUNG wire#w1
      Contact( "IO Motor MCC Panel Blending_DB"."P-30.01".QRUN )
      Coil( "Blend_T-20".IN_FBP_Transfer3 )
   END_RUNG
   RUNG wire#w1
      Contact( "IO Motor MCC Panel Blending_DB"."P-22.03".QRUN )
      Coil( "Blend_T-20".IN_FBP_CIP )
   END_RUNG
   // the same network as SCL:
   "Blend_T-20".IN_FBP_Transfer1 := "AlwaysTRUE" AND "IO Motor MCC Panel Blending_DB"."P-20.01".QRUN;
   "Blend_T-20".IN_FBP_Transfer2 := "AlwaysTRUE" AND "IO Motor MCC Panel Blending_DB"."P-21.01".QRUN;
   "Blend_T-20".IN_FBP_Transfer3 := "AlwaysTRUE" AND "IO Motor MCC Panel Blending_DB"."P-30.01".QRUN;
   "Blend_T-20".IN_FBP_CIP := "AlwaysTRUE" AND "IO Motor MCC Panel Blending_DB"."P-22.03".QRUN;
END_REGION

NETWORK
TITLE = Blending T-20 to Preparation
//to ChiliAwetan1
      O     "Blend_T-20".Dose_ChiliAwetan1.QDOSERun;  //Dose Run
      =     "Blend to Preparation"."T-20".Raw_Material.ChiliAwetan_1.DoseRun;
      O     "Blend_T-20".Dose_ChiliAwetan1.QHELD;  //Dose Held
      =     "Blend to Preparation"."T-20".Raw_Material.ChiliAwetan_1.DoseHeld;
      O     "Blend_T-20".Dose_ChiliAwetan1.QDoseComplete;  //Dose Complete
      =     "Blend to Preparation"."T-20".Raw_Material.ChiliAwetan_1.DoseComplete;
      O     "Blend_T-20".Dose_ChiliAwetan1.V_CMD;  //Valve Command
      =     "Blend to Preparation"."T-20".Raw_Material.ChiliAwetan_1.ValveCMD;
      O     "Blend_T-20".Dose_ChiliAwetan1.P_CMD;  //Pump Command
      =     "Blend to Preparation"."T-20".Raw_Material.ChiliAwetan_1.PumpCMD;
      O     "Blend_T-20".Dose.Dose_Header_Req.%X0;  //Header 1 Req
      =     "Blend to Preparation"."T-20".Raw_Material.ChiliAwetan_1.Header1_Req;
      O     "Blend_T-20".Dose.Dose_Header_Req.%X16;  //Header 2 Req
      =     "Blend to Preparation"."T-20".Raw_Material.ChiliAwetan_1.Header2_Req;
      L     "Blend to Preparation".Recipe."T-20".ChiliAwetan_1.Sp_DoseQty;  //Load Sp Dose From Recipe
      T     "Blend_T-20".SP_ChiliAwetan1.Dose_SP;
      L     "Blend_T-20".Dose_ChiliAwetan1.P_SPEED;  //Pump Speed
      T     "Blend to Preparation".Recipe."T-20".ChiliAwetan_1.SP_PumpSpeed;

//to ChiliAwetan2
      O     "Blend_T-20".Dose_ChiliAwetan2.QDOSERun;  //Dose Run
      =     "Blend to Preparation"."T-20".Raw_Material.ChiliAwetan_2.DoseRun;
      O     "Blend_T-20".Dose_ChiliAwetan2.QHELD;  //Dose Held
      =     "Blend to Preparation"."T-20".Raw_Material.ChiliAwetan_2.DoseHeld;
      O     "Blend_T-20".Dose_ChiliAwetan2.QDoseComplete;  //Dose Complete
      =     "Blend to Preparation"."T-20".Raw_Material.ChiliAwetan_2.DoseComplete;
      O     "Blend_T-20".Dose_ChiliAwetan2.V_CMD;  //Valve Command
      =     "Blend to Preparation"."T-20".Raw_Material.ChiliAwetan_2.ValveCMD;
      O     "Blend_T-20".Dose_ChiliAwetan2.P_CMD;  //Pump Command
      =     "Blend to Preparation"."T-20".Raw_Material.ChiliAwetan_2.PumpCMD;
      O     "Blend_T-20".Dose.Dose_Header_Req.%X1;  //Header 1 Req
      =     "Blend to Preparation"."T-20".Raw_Material.ChiliAwetan_2.Header1_Req;
      O     "Blend_T-20".Dose.Dose_Header_Req.%X17;  //Header 2 Req
      =     "Blend to Preparation"."T-20".Raw_Material.ChiliAwetan_2.Header2_Req;
      L     "Blend to Preparation".Recipe."T-20".ChiliAwetan_2.Sp_DoseQty;  //Load Sp Dose From Recipe
      T     "Blend_T-20".SP_ChiliAwetan2.Dose_SP;
      L     "Blend_T-20".Dose_ChiliAwetan2.P_SPEED;  //Pump Speed
      T     "Blend to Preparation".Recipe."T-20".ChiliAwetan_2.SP_PumpSpeed;

//to ChiliAwetan3
      O     "Blend_T-20".Dose_ChiliAwetan3.QDOSERun;  //Dose Run
      =     "Blend to Preparation"."T-20".Raw_Material.ChiliAwetan_3.DoseRun;
      O     "Blend_T-20".Dose_ChiliAwetan3.QHELD;  //Dose Held
      =     "Blend to Preparation"."T-20".Raw_Material.ChiliAwetan_3.DoseHeld;
      O     "Blend_T-20".Dose_ChiliAwetan3.QDoseComplete;  //Dose Complete
      =     "Blend to Preparation"."T-20".Raw_Material.ChiliAwetan_3.DoseComplete;
      O     "Blend_T-20".Dose_ChiliAwetan3.V_CMD;  //Valve Command
      =     "Blend to Preparation"."T-20".Raw_Material.ChiliAwetan_3.ValveCMD;
      O     "Blend_T-20".Dose_ChiliAwetan3.P_CMD;  //Pump Command
      =     "Blend to Preparation"."T-20".Raw_Material.ChiliAwetan_3.PumpCMD;
      O     "Blend_T-20".Dose.Dose_Header_Req.%X2;  //Header 1 Req
      =     "Blend to Preparation"."T-20".Raw_Material.ChiliAwetan_3.Header1_Req;
      O     "Blend_T-20".Dose.Dose_Header_Req.%X18;  //Header 2 Req
      =     "Blend to Preparation"."T-20".Raw_Material.ChiliAwetan_3.Header2_Req;
      L     "Blend to Preparation".Recipe."T-20".ChiliAwetan_3.Sp_DoseQty;  //Load Sp Dose From Recipe
      T     "Blend_T-20".SP_ChiliAwetan3.Dose_SP;
      L     "Blend_T-20".Dose_ChiliAwetan3.P_SPEED;  //Pump Speed
      T     "Blend to Preparation".Recipe."T-20".ChiliAwetan_3.SP_PumpSpeed;

//to Tomato
      O     "Blend_T-20".Dose_Tomato.QDOSERun;  //Dose Run
      =     "Blend to Preparation"."T-20".Raw_Material.Tomato.DoseRun;
      O     "Blend_T-20".Dose_Tomato.QHELD;  //Dose Held
      =     "Blend to Preparation"."T-20".Raw_Material.Tomato.DoseHeld;
      O     "Blend_T-20".Dose_Tomato.QDoseComplete;  //Dose Complete
      =     "Blend to Preparation"."T-20".Raw_Material.Tomato.DoseComplete;
      O     "Blend_T-20".Dose_Tomato.V_CMD;  //Valve Command
      =     "Blend to Preparation"."T-20".Raw_Material.Tomato.ValveCMD;
      O     "Blend_T-20".Dose_Tomato.P_CMD;  //Pump Command
      =     "Blend to Preparation"."T-20".Raw_Material.Tomato.PumpCMD;
      O     "Blend_T-20".Dose.Dose_Header_Req.%X3;  //Header 1 Req
      =     "Blend to Preparation"."T-20".Raw_Material.Tomato.Header1_Req;
      O     "Blend_T-20".Dose.Dose_Header_Req.%X19;  //Header 2 Req
      =     "Blend to Preparation"."T-20".Raw_Material.Tomato.Header2_Req;
      L     "Blend to Preparation".Recipe."T-20".Tomato.Sp_DoseQty;  //Load Sp Dose From Recipe
      T     "Blend_T-20".SP_Tomato.Dose_SP;
      L     "Blend_T-20".Dose_Tomato.P_SPEED;  //Pump Speed
      T     "Blend to Preparation".Recipe."T-20".Tomato.SP_PumpSpeed;

//to ChiliFresh1
      O     "Blend_T-20".Dose_ChiliFresh1.QDOSERun;  //Dose Run
      =     "Blend to Preparation"."T-20".Raw_Material.ChiliFresh_1.DoseRun;
      O     "Blend_T-20".Dose_ChiliFresh1.QHELD;  //Dose Held
      =     "Blend to Preparation"."T-20".Raw_Material.ChiliFresh_1.DoseHeld;
      O     "Blend_T-20".Dose_ChiliFresh1.QDoseComplete;  //Dose Complete
      =     "Blend to Preparation"."T-20".Raw_Material.ChiliFresh_1.DoseComplete;
      O     "Blend_T-20".Dose_ChiliFresh1.V_CMD;  //Valve Command
      =     "Blend to Preparation"."T-20".Raw_Material.ChiliFresh_1.ValveCMD;
      O     "Blend_T-20".Dose_ChiliFresh1.P_CMD;  //Pump Command
      =     "Blend to Preparation"."T-20".Raw_Material.ChiliFresh_1.PumpCMD;
      O     "Blend_T-20".Dose.Dose_Header_Req.%X4;  //Header 1 Req
      =     "Blend to Preparation"."T-20".Raw_Material.ChiliFresh_1.Header1_Req;
      O     "Blend_T-20".Dose.Dose_Header_Req.%X20;  //Header 2 Req
      =     "Blend to Preparation"."T-20".Raw_Material.ChiliFresh_1.Header2_Req;
      L     "Blend to Preparation".Recipe."T-20".ChiliFresh_1.Sp_DoseQty;  //Load Sp Dose From Recipe
      T     "Blend_T-20".SP_ChiliFresh1.Dose_SP;
      L     "Blend_T-20".Dose_ChiliFresh1.P_SPEED;  //Pump Speed
      T     "Blend to Preparation".Recipe."T-20".ChiliFresh_1.SP_PumpSpeed;

//to ChiliFresh2
      O     "Blend_T-20".Dose_ChiliFresh2.QDOSERun;  //Dose Run
      =     "Blend to Preparation"."T-20".Raw_Material.ChiliFresh_2.DoseRun;
      O     "Blend_T-20".Dose_ChiliFresh2.QHELD;  //Dose Held
      =     "Blend to Preparation"."T-20".Raw_Material.ChiliFresh_2.DoseHeld;
      O     "Blend_T-20".Dose_ChiliFresh2.QDoseComplete;  //Dose Complete
      =     "Blend to Preparation"."T-20".Raw_Material.ChiliFresh_2.DoseComplete;
      O     "Blend_T-20".Dose_ChiliFresh2.V_CMD;  //Valve Command
      =     "Blend to Preparation"."T-20".Raw_Material.ChiliFresh_2.ValveCMD;
      O     "Blend_T-20".Dose_ChiliFresh2.P_CMD;  //Pump Command
      =     "Blend to Preparation"."T-20".Raw_Material.ChiliFresh_2.PumpCMD;
      O     "Blend_T-20".Dose.Dose_Header_Req.%X5;  //Header 1 Req
      =     "Blend to Preparation"."T-20".Raw_Material.ChiliFresh_2.Header1_Req;
      O     "Blend_T-20".Dose.Dose_Header_Req.%X21;  //Header 2 Req
      =     "Blend to Preparation"."T-20".Raw_Material.ChiliFresh_2.Header2_Req;
      L     "Blend to Preparation".Recipe."T-20".ChiliFresh_2.Sp_DoseQty;  //Load Sp Dose From Recipe
      T     "Blend_T-20".SP_ChiliFresh2.Dose_SP;
      L     "Blend_T-20".Dose_ChiliFresh2.P_SPEED;  //Pump Speed
      T     "Blend to Preparation".Recipe."T-20".ChiliFresh_2.SP_PumpSpeed;

//to ChiliFresh3
      O     "Blend_T-20".Dose_ChiliFresh3.QDOSERun;  //Dose Run
      =     "Blend to Preparation"."T-20".Raw_Material.ChiliFresh_3.DoseRun;
      O     "Blend_T-20".Dose_ChiliFresh3.QHELD;  //Dose Held
      =     "Blend to Preparation"."T-20".Raw_Material.ChiliFresh_3.DoseHeld;
      O     "Blend_T-20".Dose_ChiliFresh3.QDoseComplete;  //Dose Complete
      =     "Blend to Preparation"."T-20".Raw_Material.ChiliFresh_3.DoseComplete;
      O     "Blend_T-20".Dose_ChiliFresh3.V_CMD;  //Valve Command
      =     "Blend to Preparation"."T-20".Raw_Material.ChiliFresh_3.ValveCMD;
      O     "Blend_T-20".Dose_ChiliFresh3.P_CMD;  //Pump Command
      =     "Blend to Preparation"."T-20".Raw_Material.ChiliFresh_3.PumpCMD;
      O     "Blend_T-20".Dose.Dose_Header_Req.%X6;  //Header 1 Req
      =     "Blend to Preparation"."T-20".Raw_Material.ChiliFresh_3.Header1_Req;
      O     "Blend_T-20".Dose.Dose_Header_Req.%X22;  //Header 2 Req
      =     "Blend to Preparation"."T-20".Raw_Material.ChiliFresh_3.Header2_Req;
      L     "Blend to Preparation".Recipe."T-20".ChiliFresh_3.Sp_DoseQty;  //Load Sp Dose From Recipe
      T     "Blend_T-20".SP_ChiliFresh3.Dose_SP;
      L     "Blend_T-20".Dose_ChiliFresh3.P_SPEED;  //Pump Speed
      T     "Blend to Preparation".Recipe."T-20".ChiliFresh_3.SP_PumpSpeed;

//to Garlic
      O     "Blend_T-20".Dose_Garlic.QDOSERun;  //Dose Run
      =     "Blend to Preparation"."T-20".Raw_Material.Garlic.DoseRun;
      O     "Blend_T-20".Dose_Garlic.QHELD;  //Dose Held
      =     "Blend to Preparation"."T-20".Raw_Material.Garlic.DoseHeld;
      O     "Blend_T-20".Dose_Garlic.QDoseComplete;  //Dose Complete
      =     "Blend to Preparation"."T-20".Raw_Material.Garlic.DoseComplete;
      O     "Blend_T-20".Dose_Garlic.V_CMD;  //Valve Command
      =     "Blend to Preparation"."T-20".Raw_Material.Garlic.ValveCMD;
      O     "Blend_T-20".Dose_Garlic.P_CMD;  //Pump Command
      =     "Blend to Preparation"."T-20".Raw_Material.Garlic.PumpCMD;
      O     "Blend_T-20".Dose.Dose_Header_Req.%X7;  //Header 1 Req
      =     "Blend to Preparation"."T-20".Raw_Material.Garlic.Header1_Req;
      O     "Blend_T-20".Dose.Dose_Header_Req.%X23;  //Header 2 Req
      =     "Blend to Preparation"."T-20".Raw_Material.Garlic.Header2_Req;
      L     "Blend to Preparation".Recipe."T-20".Garlic.Sp_DoseQty;  //Load Sp Dose From Recipe
      T     "Blend_T-20".SP_Garlic.Dose_SP;
      L     "Blend_T-20".Dose_Garlic.P_SPEED;  //Pump Speed
      T     "Blend to Preparation".Recipe."T-20".Garlic.SP_PumpSpeed;

//to Vinegar
      O     "Blend_T-20".Dose_Vinegar.QDOSERun;  //Dose Run
      =     "Blend to Preparation"."T-20".Raw_Material.Vinegar.DoseRun;
      O     "Blend_T-20".Dose_Vinegar.QHELD;  //Dose Held
      =     "Blend to Preparation"."T-20".Raw_Material.Vinegar.DoseHeld;
      O     "Blend_T-20".Dose_Vinegar.QDoseComplete;  //Dose Complete
      =     "Blend to Preparation"."T-20".Raw_Material.Vinegar.DoseComplete;
      O     "Blend_T-20".Dose_Vinegar.V_CMD;  //Valve Command
      =     "Blend to Preparation"."T-20".Raw_Material.Vinegar.ValveCMD;
      O     "Blend_T-20".Dose_Vinegar.P_CMD;  //Pump Command
      =     "Blend to Preparation"."T-20".Raw_Material.Vinegar.PumpCMD;
      L     "Blend to Preparation".Recipe."T-20".Vinegar.Sp_DoseQty;  //Load Sp Dose From Recipe
      T     "Blend_T-20".SP_Vinegar.Dose_SP;
      L     "Blend_T-20".Dose_Vinegar.P_SPEED;  //Pump Speed
      T     "Blend to Preparation".Recipe."T-20".Vinegar.SP_PumpSpeed;

//to HW
      O     "Blend_T-20".Dose_HW.QDOSERun;  //Dose Run
      =     "Blend to Preparation"."T-20".Raw_Material.HW.DoseRun;
      O     "Blend_T-20".Dose_HW.QHELD;  //Dose Held
      =     "Blend to Preparation"."T-20".Raw_Material.HW.DoseHeld;
      O     "Blend_T-20".Dose_HW.QDoseComplete;  //Dose Complete
      =     "Blend to Preparation"."T-20".Raw_Material.HW.DoseComplete;
      O     "Blend_T-20".Dose_HW.V_CMD;  //Valve Command
      =     "Blend to Preparation"."T-20".Raw_Material.HW.ValveCMD;
      O     "Blend_T-20".Dose_HW.P_CMD;  //Pump Command
      =     "Blend to Preparation"."T-20".Raw_Material.HW.PumpCMD;
      O     "Blend_T-20".Dose.Dose_Header_Req.%X8;  //Header 1 Req
      =     "Blend to Preparation"."T-20".Raw_Material.HW.Header1_Req;
      O     "Blend_T-20".Dose.Dose_Header_Req.%X24;  //Header 2 Req
      =     "Blend to Preparation"."T-20".Raw_Material.HW.Header2_Req;

      L     "Blend to Preparation".Recipe."T-20".HW.Sp_Flush_to_BlendQty;  //Load Flush to Blend Sp Dose From Recipe
      T     "Blend_T-20"."HW Flushing".Qty."Flush to Blend Qty";
      L     "Blend to Preparation".Recipe."T-20".HW.Sp_Flush_to_DrainQty;  //Load Flush to Blend Sp Dose From Recipe
      T     "Blend_T-20"."HW Flushing".Qty."Flush to Drain Qty";  //Load Drain Time from recipe
      L     "Blend to Preparation".Recipe."T-20".HW.Sp_DrainTime;
      T     "Blend_T-20"."HW Flushing".TimeDrain_SP;

      L     "Blend_T-20".Dose_HW.P_SPEED;  //Pump Speed
      T     "Blend to Preparation".Recipe."T-20".HW.SP_PumpSpeed;

//General
      O     "Blend_T-20".IN_FBAV_Header1;
      =     "Blend to Preparation"."T-20".LineHeader1_OK;
      O     "Blend_T-20".IN_FBAV_Header2;
      =     "Blend to Preparation"."T-20".LineHeader2_OK;
      O     "Blend_T-20".IN_FBAV_Vinegar;
      =     "Blend to Preparation"."T-20".LineVinegar_OK;


NETWORK
TITLE = ChiliAwetan1 to Blending T-21
//Valve Open
      A     "Preparation to Blend"."T-02_ChiliAwetan_1".Valve_Open;
      A(;
      O(;
      A     "Blend_T-21".Dose.Dose_Header_Req.%X0;
      A     "Blend_T-21".IN_FBAV_Header1;
      );
      O(;
      A     "Blend_T-21".Dose.Dose_Header_Req.%X16;
      A     "Blend_T-21".IN_FBAV_Header2;
      );
      );
      =     "Blend_T-21".Dose_ChiliAwetan1.V_OPEN;
//Pump On
      O     "Preparation to Blend"."T-02_ChiliAwetan_1".Pump_Run;
      =     "Blend_T-21".Dose_ChiliAwetan1.P_RUN;
//Tank Available
      O     "Preparation to Blend"."T-02_ChiliAwetan_1".Tank_Available;
      O     "Blend_T-21".Dose_ChiliAwetan1.QDOSERun;
      =     "Blend_T-21".Dose.Dose_Tank_Available.%X0;
//Product Ready
      O     "Preparation to Blend"."T-02_ChiliAwetan_1".Product_Ready;
      =     "Blend_T-21".Dose.Dose_Prod_Ready.%X0;
//Level Tank
      L     "Preparation to Blend"."T-02_ChiliAwetan_1".Level;
      T     "Blend_T-21"."Dose_Level_%"."ChiliAwetan1%";


NETWORK
TITLE = ChiliAwetan2 to Blending T-21
//Valve Open
      A     "Preparation to Blend"."T-03_ChiliAwetan_2".Valve_Open;
      A(;
      O(;
      A     "Blend_T-21".Dose.Dose_Header_Req.%X1;
      A     "Blend_T-21".IN_FBAV_Header1;
      );
      O(;
      A     "Blend_T-21".Dose.Dose_Header_Req.%X17;
      A     "Blend_T-21".IN_FBAV_Header2;
      );
      );
      =     "Blend_T-21".Dose_ChiliAwetan2.V_OPEN;
//Pump On
      O     "Preparation to Blend"."T-03_ChiliAwetan_2".Pump_Run;
      =     "Blend_T-21".Dose_ChiliAwetan2.P_RUN;
//Tank Available
      O     "Preparation to Blend"."T-03_ChiliAwetan_2".Tank_Available;
      O     "Blend_T-21".Dose_ChiliAwetan2.QDOSERun;
      =     "Blend_T-21".Dose.Dose_Tank_Available.%X1;
//Product Ready
      O     "Preparation to Blend"."T-03_ChiliAwetan_2".Product_Ready;
      =     "Blend_T-21".Dose.Dose_Prod_Ready.%X1;
//Level Tank
      L     "Preparation to Blend"."T-03_ChiliAwetan_2".Level;
      T     "Blend_T-21"."Dose_Level_%"."ChiliAwetan2%";


NETWORK
TITLE = ChiliAwetan3 to Blending T-21
//Valve Open
      A     "Preparation to Blend"."T-04_ChiliAwetan_3".Valve_Open;
      A(;
      O(;
      A     "Blend_T-21".Dose.Dose_Header_Req.%X2;
      A     "Blend_T-21".IN_FBAV_Header1;
      );
      O(;
      A     "Blend_T-21".Dose.Dose_Header_Req.%X18;
      A     "Blend_T-21".IN_FBAV_Header2;
      );
      );
      =     "Blend_T-21".Dose_ChiliAwetan3.V_OPEN;
//Pump On
      O     "Preparation to Blend"."T-04_ChiliAwetan_3".Pump_Run;
      =     "Blend_T-21".Dose_ChiliAwetan3.P_RUN;
//Tank Available
      O     "Preparation to Blend"."T-04_ChiliAwetan_3".Tank_Available;
      O     "Blend_T-21".Dose_ChiliAwetan3.QDOSERun;
      =     "Blend_T-21".Dose.Dose_Tank_Available.%X2;
//Product Ready
      O     "Preparation to Blend"."T-04_ChiliAwetan_3".Product_Ready;
      =     "Blend_T-21".Dose.Dose_Prod_Ready.%X2;
//Level Tank
      L     "Preparation to Blend"."T-04_ChiliAwetan_3".Level;
      T     "Blend_T-21"."Dose_Level_%"."ChiliAwetan3%";


NETWORK
TITLE = Tomato to Blending T-21
//Valve Open
      A     "Preparation to Blend"."T-05_Tomato".Valve_Open;
      A(;
      O(;
      A     "Blend_T-21".Dose.Dose_Header_Req.%X3;
      A     "Blend_T-21".IN_FBAV_Header1;
      );
      O(;
      A     "Blend_T-21".Dose.Dose_Header_Req.%X19;
      A     "Blend_T-21".IN_FBAV_Header2;
      );
      );
      =     "Blend_T-21".Dose_Tomato.V_OPEN;
//Pump On
      O     "Preparation to Blend"."T-05_Tomato".Pump_Run;
      =     "Blend_T-21".Dose_Tomato.P_RUN;
//Tank Available
      O     "Preparation to Blend"."T-05_Tomato".Tank_Available;
      O     "Blend_T-21".Dose_Tomato.QDOSERun;
      =     "Blend_T-21".Dose.Dose_Tank_Available.%X3;
//Product Ready
      O     "Preparation to Blend"."T-05_Tomato".Product_Ready;
      =     "Blend_T-21".Dose.Dose_Prod_Ready.%X3;
//Level Tank
      L     "Preparation to Blend"."T-05_Tomato".Level;
      T     "Blend_T-21"."Dose_Level_%"."Tomato%";


NETWORK
TITLE = ChiliFresh1 to Blending T-21
//Valve Open
      A     "Preparation to Blend"."T-06_ChiliFresh_1".Valve_Open;
      A(;
      O(;
      A     "Blend_T-21".Dose.Dose_Header_Req.%X4;
      A     "Blend_T-21".IN_FBAV_Header1;
      );
      O(;
      A     "Blend_T-21".Dose.Dose_Header_Req.%X20;
      A     "Blend_T-21".IN_FBAV_Header2;
      );
      );
      =     "Blend_T-21".Dose_ChiliFresh1.V_OPEN;
//Pump On
      O     "Preparation to Blend"."T-06_ChiliFresh_1".Pump_Run;
      =     "Blend_T-21".Dose_ChiliFresh1.P_RUN;
//Tank Available
      O     "Preparation to Blend"."T-06_ChiliFresh_1".Tank_Available;
      O     "Blend_T-21".Dose_ChiliFresh1.QDOSERun;
      =     "Blend_T-21".Dose.Dose_Tank_Available.%X4;
//Product Ready
      O     "Preparation to Blend"."T-06_ChiliFresh_1".Product_Ready;
      =     "Blend_T-21".Dose.Dose_Prod_Ready.%X4;
//Level Tank
      L     "Preparation to Blend"."T-06_ChiliFresh_1".Level;
      T     "Blend_T-21"."Dose_Level_%"."ChiliFresh1%";


NETWORK
TITLE = ChiliFresh2 to Blending T-21
//Valve Open
      A     "Preparation to Blend"."T-07_ChiliFresh_2".Valve_Open;
      A(;
      O(;
      A     "Blend_T-21".Dose.Dose_Header_Req.%X5;
      A     "Blend_T-21".IN_FBAV_Header1;
      );
      O(;
      A     "Blend_T-21".Dose.Dose_Header_Req.%X21;
      A     "Blend_T-21".IN_FBAV_Header2;
      );
      );
      =     "Blend_T-21".Dose_ChiliFresh2.V_OPEN;
//Pump On
      O     "Preparation to Blend"."T-07_ChiliFresh_2".Pump_Run;
      =     "Blend_T-21".Dose_ChiliFresh2.P_RUN;
//Tank Available
      O     "Preparation to Blend"."T-07_ChiliFresh_2".Tank_Available;
      O     "Blend_T-21".Dose_ChiliFresh2.QDOSERun;
      =     "Blend_T-21".Dose.Dose_Tank_Available.%X5;
//Product Ready
      O     "Preparation to Blend"."T-07_ChiliFresh_2".Product_Ready;
      =     "Blend_T-21".Dose.Dose_Prod_Ready.%X5;
//Level Tank
      L     "Preparation to Blend"."T-07_ChiliFresh_2".Level;
      T     "Blend_T-21"."Dose_Level_%"."ChiliFresh2%";


NETWORK
TITLE = ChiliFresh3 to Blending T-21
//Valve Open
      A     "Preparation to Blend"."T-08_ChiliFresh_3".Valve_Open;
      A(;
      O(;
      A     "Blend_T-21".Dose.Dose_Header_Req.%X6;
      A     "Blend_T-21".IN_FBAV_Header1;
      );
      O(;
      A     "Blend_T-21".Dose.Dose_Header_Req.%X22;
      A     "Blend_T-21".IN_FBAV_Header2;
      );
      );
      =     "Blend_T-21".Dose_ChiliFresh3.V_OPEN;
//Pump On
      O     "Preparation to Blend"."T-08_ChiliFresh_3".Pump_Run;
      =     "Blend_T-21".Dose_ChiliFresh3.P_RUN;
//Tank Available
      O     "Preparation to Blend"."T-08_ChiliFresh_3".Tank_Available;
      O     "Blend_T-21".Dose_ChiliFresh3.QDOSERun;
      =     "Blend_T-21".Dose.Dose_Tank_Available.%X6;
//Product Ready
      O     "Preparation to Blend"."T-08_ChiliFresh_3".Product_Ready;
      =     "Blend_T-21".Dose.Dose_Prod_Ready.%X6;
//Level Tank
      L     "Preparation to Blend"."T-08_ChiliFresh_3".Level;
      T     "Blend_T-21"."Dose_Level_%"."ChiliFresh3%";


NETWORK
TITLE = Garlic to Blending T-21
//Valve Open
      A     "Preparation to Blend"."T-09_Garlic".Valve_Open;
      A(;
      O(;
      A     "Blend_T-21".Dose.Dose_Header_Req.%X7;
      A     "Blend_T-21".IN_FBAV_Header1;
      );
      O(;
      A     "Blend_T-21".Dose.Dose_Header_Req.%X23;
      A     "Blend_T-21".IN_FBAV_Header2;
      );
      );
      =     "Blend_T-21".Dose_Garlic.V_OPEN;
//Pump On
      O     "Preparation to Blend"."T-09_Garlic".Pump_Run;
      =     "Blend_T-21".Dose_Garlic.P_RUN;
//Tank Available
      O     "Preparation to Blend"."T-09_Garlic".Tank_Available;
      O     "Blend_T-21".Dose_Garlic.QDOSERun;
      =     "Blend_T-21".Dose.Dose_Tank_Available.%X7;
//Product Ready
      O     "Preparation to Blend"."T-09_Garlic".Product_Ready;
      =     "Blend_T-21".Dose.Dose_Prod_Ready.%X7;
//Level Tank
      L     "Preparation to Blend"."T-09_Garlic".Level;
      T     "Blend_T-21"."Dose_Level_%"."Garlic%";


NETWORK
TITLE = Vinegar to Blending T-21
//Valve Open
      A     "Preparation to Blend"."T-10_Vinegar".Valve_Open;
      A     "Blend_T-21".IN_FBAV_Vinegar;
      =     "Blend_T-21".Dose_Vinegar.V_OPEN;
//Pump On
      O     "Preparation to Blend"."T-10_Vinegar".Pump_Run;
      =     "Blend_T-21".Dose_Vinegar.P_RUN;
//Tank Available
      O     "Preparation to Blend"."T-10_Vinegar".Tank_Available;
      O     "Blend_T-21".Dose_Vinegar.QDOSERun;
      =     "Blend_T-21".Dose.Dose_Tank_Available.%X9;
//Product Ready
      O     "Preparation to Blend"."T-10_Vinegar".Product_Ready;
      =     "Blend_T-21".Dose.Dose_Prod_Ready.%X9;
//Level Tank
      L     "Preparation to Blend"."T-10_Vinegar".Level;
      T     "Blend_T-21"."Dose_Level_%"."Vinegar%";


NETWORK
TITLE = HW to Blending T-21
//Valve Open
      A     "Preparation to Blend"."T-51_HW".Valve_Open;
      A(;
      O(;
      A     "Blend_T-21".Dose.Dose_Header_Req.%X8;
      A     "Blend_T-21".IN_FBAV_Header1;
      );
      O(;
      A     "Blend_T-21".Dose.Dose_Header_Req.%X24;
      A     "Blend_T-21".IN_FBAV_Header2;
      );
      );
      =     "Blend_T-21".Dose_HW.V_OPEN;
//Pump On
      O     "Preparation to Blend"."T-51_HW".Pump_Run;
      =     "Blend_T-21".Dose_HW.P_RUN;
//Tank Available
      O     "Preparation to Blend"."T-51_HW".Tank_Available;
      O     "Blend_T-21".Dose_HW.QDOSERun;
      =     "Blend_T-21".Dose.Dose_Tank_Available.%X8;
//Product Ready
      O     "Preparation to Blend"."T-51_HW".Product_Ready;
      =     "Blend_T-21".Dose.Dose_Prod_Ready.%X8;
//Level Tank
// L     "Preparation to Blend"."T-01_HW".Level
// T     "Blend_T-21"."Dose_Level_%"."HW%"


REGION Network 35: Homomixer 12.00 to Blending T-21.00
   RUNG wire#powerrail
      Contact( "AlwaysTRUE" )
      wire#w1
      Contact( "IO Valve Homomixer_DB"."AV-12.03".FB_OPEN )
      Contact( "Blend_T-21".IN_FBAV_Homomixer )
      Coil( "Blend_T-21".Dose_Homomixer.V_OPEN )
   END_RUNG
   RUNG wire#w1
      Contact( "IO Valve Homomixer_DB"."P-12.01".FB_ON )
      Coil( "Blend_T-21".Dose_Homomixer.P_RUN )
   END_RUNG
   RUNG wire#w1
      Contact( "T-12.00_Homomixer".Out_Tank_Ready )
      wire#w2
      Coil( "Blend_T-21".Dose.Dose_Tank_Available.%X13 )
   END_RUNG
   RUNG wire#w1
      Contact( "Blend_T-21".Dose_Homomixer.QDOSERun )
   END_RUNG wire#w2
   RUNG wire#w1
      Contact( "T-12.00_Homomixer".Out_Prod_Ready )
      Coil( "Blend_T-21".Dose.Dose_Prod_Ready.%X13 )
   END_RUNG
   // the same network as SCL:
   "Blend_T-21".Dose_Homomixer.V_OPEN := "AlwaysTRUE" AND "IO Valve Homomixer_DB"."AV-12.03".FB_OPEN AND "Blend_T-21".IN_FBAV_Homomixer;
   "Blend_T-21".Dose_Homomixer.P_RUN := "AlwaysTRUE" AND "IO Valve Homomixer_DB"."P-12.01".FB_ON;
   "Blend_T-21".Dose.Dose_Tank_Available.%X13 := "AlwaysTRUE" AND ("T-12.00_Homomixer".Out_Tank_Ready OR "Blend_T-21".Dose_Homomixer.QDOSERun);
   "Blend_T-21".Dose.Dose_Prod_Ready.%X13 := "AlwaysTRUE" AND "T-12.00_Homomixer".Out_Prod_Ready;
END_REGION

REGION Network 36: Sugar to Blending T-21
   RUNG wire#powerrail
      Contact( "AlwaysTRUE" )
      wire#w1
      Contact( "Sugar to Mix"."System ready to run" )
      wire#w2
      Coil( "Blend_T-21".Dose.Dose_Tank_Available.%X10 )
   END_RUNG
   RUNG wire#w1
      Contact( "Blend_T-21".Dose_Sugar.QDOSERun )
   END_RUNG wire#w2
   RUNG wire#w1
      Contact( "Sugar to Mix"."System ready to run" )
      Coil( "Blend_T-21".Dose.Dose_Prod_Ready.%X10 )
   END_RUNG
   RUNG wire#w1
      Contact( "Blend_T-21".Dose_Sugar.QDOSERun )
      Contact( "Sugar to Mix"."Transfer in process" )
      Coil( "General_Blend".Sugar."In Process"."T-21" )
   END_RUNG
   RUNG wire#w1
      Move(in := "Blend to Preparation".Recipe."T-21".Sugar.Sp_DoseQty, out1 => "Blend_T-21".SP_Sugar.Dose_SP)
   END_RUNG
   // the same network as SCL:
   "Blend_T-21".Dose.Dose_Tank_Available.%X10 := "AlwaysTRUE" AND ("Sugar to Mix"."System ready to run" OR "Blend_T-21".Dose_Sugar.QDOSERun);
   "Blend_T-21".Dose.Dose_Prod_Ready.%X10 := "AlwaysTRUE" AND "Sugar to Mix"."System ready to run";
   "General_Blend".Sugar."In Process"."T-21" := "AlwaysTRUE" AND "Blend_T-21".Dose_Sugar.QDOSERun AND "Sugar to Mix"."Transfer in process";
   IF "AlwaysTRUE" THEN
       "Blend_T-21".SP_Sugar.Dose_SP := "Blend to Preparation".Recipe."T-21".Sugar.Sp_DoseQty;
   END_IF;
END_REGION

REGION Network 37: Salt to Blending T-21
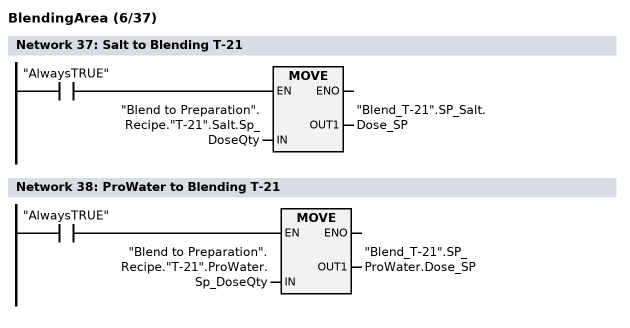
   RUNG wire#powerrail
      Contact( "AlwaysTRUE" )
      Move(in := "Blend to Preparation".Recipe."T-21".Salt.Sp_DoseQty, out1 => "Blend_T-21".SP_Salt.Dose_SP)
   END_RUNG
   // the same network as SCL:
   IF "AlwaysTRUE" THEN
       "Blend_T-21".SP_Salt.Dose_SP := "Blend to Preparation".Recipe."T-21".Salt.Sp_DoseQty;
   END_IF;
END_REGION

REGION Network 38: ProWater to Blending T-21
   RUNG wire#powerrail
      Contact( "AlwaysTRUE" )
      Move(in := "Blend to Preparation".Recipe."T-21".ProWater.Sp_DoseQty, out1 => "Blend_T-21".SP_ProWater.Dose_SP)
   END_RUNG
   // the same network as SCL:
   IF "AlwaysTRUE" THEN
       "Blend_T-21".SP_ProWater.Dose_SP := "Blend to Preparation".Recipe."T-21".ProWater.Sp_DoseQty;
   END_IF;
END_REGION

REGION Network 39: Blending T-21
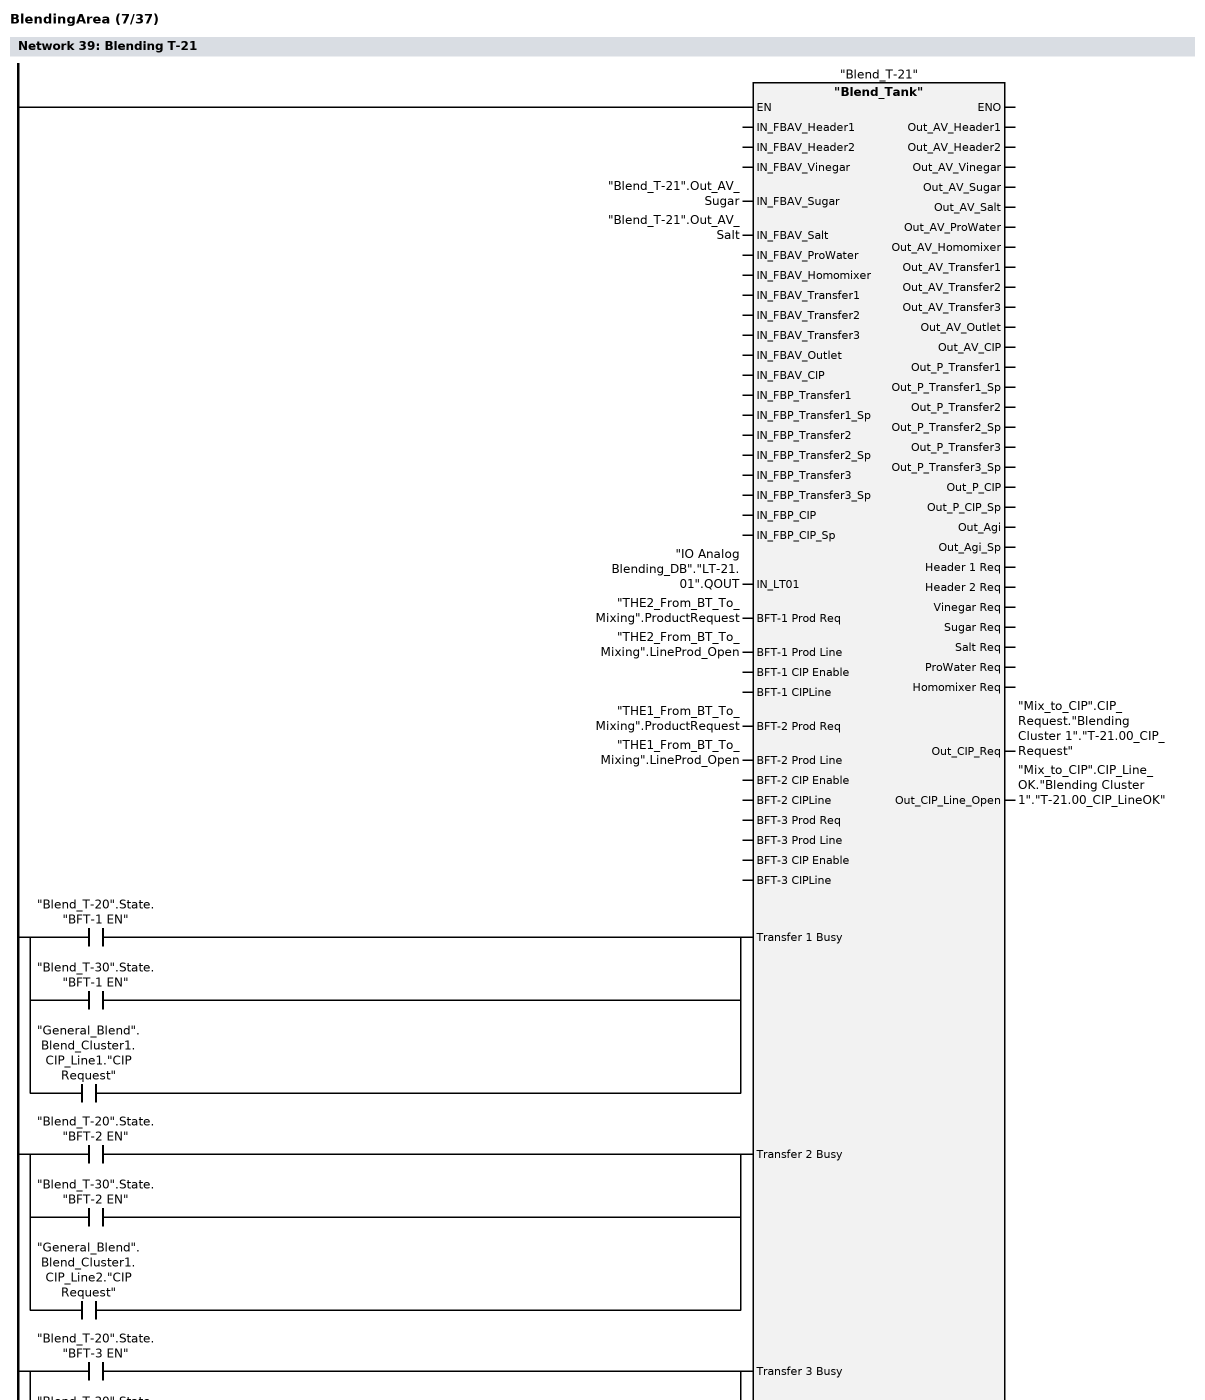
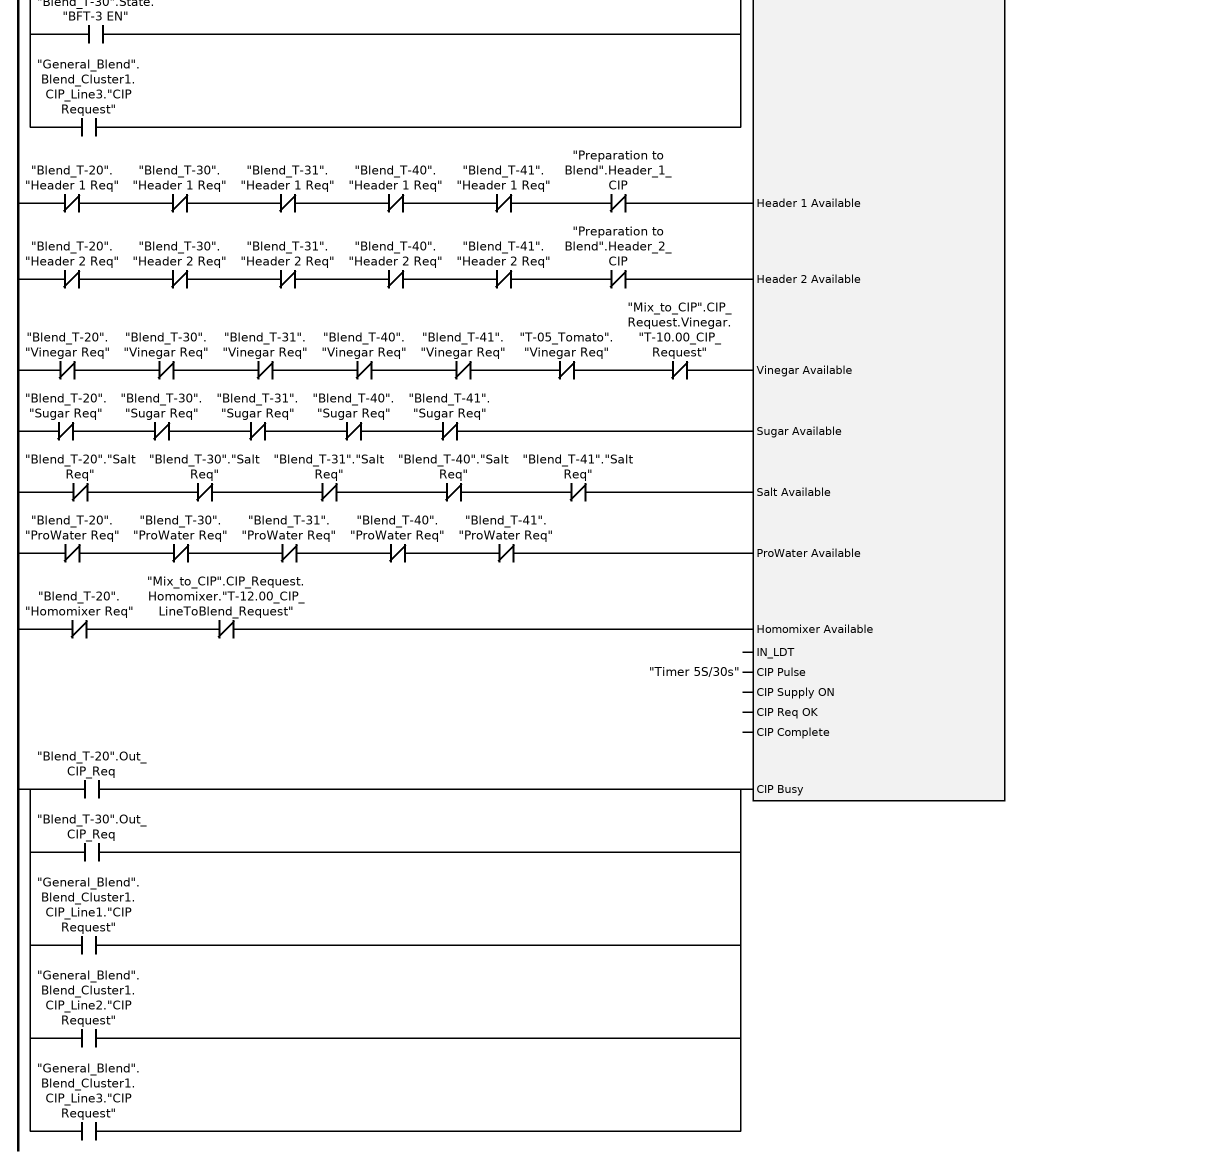
   RUNG wire#powerrail
      "Blend_T-21"("Transfer 1 Busy" := wire#w1, "Transfer 2 Busy" := wire#w2, "Transfer 3 Busy" := wire#w3, "Header 1 Available" := wire#w4, "Header 2 Available" := wire#w5, "Vinegar Available" := wire#w6, "Sugar Available" := wire#w7, "Salt Available" := wire#w8, "ProWater Available" := wire#w9, "Homomixer Available" := wire#w10, "CIP Busy" := wire#w11, IN_FBAV_Header1 :=, IN_FBAV_Header2 :=, IN_FBAV_Vinegar :=, IN_FBAV_Sugar := "Blend_T-21".Out_AV_Sugar, IN_FBAV_Salt := "Blend_T-21".Out_AV_Salt, IN_FBAV_ProWater :=, IN_FBAV_Homomixer :=, IN_FBAV_Transfer1 :=, IN_FBAV_Transfer2 :=, IN_FBAV_Transfer3 :=, IN_FBAV_Outlet :=, IN_FBAV_CIP :=, IN_FBP_Transfer1 :=, IN_FBP_Transfer1_Sp :=, IN_FBP_Transfer2 :=, IN_FBP_Transfer2_Sp :=, IN_FBP_Transfer3 :=, IN_FBP_Transfer3_Sp :=, IN_FBP_CIP :=, IN_FBP_CIP_Sp :=, IN_LT01 := "IO Analog Blending_DB"."LT-21.01".QOUT, "BFT-1 Prod Req" := "THE2_From_BT_To_Mixing".ProductRequest, "BFT-1 Prod Line" := "THE2_From_BT_To_Mixing".LineProd_Open, "BFT-1 CIP Enable" :=, "BFT-1 CIPLine" :=, "BFT-2 Prod Req" := "THE1_From_BT_To_Mixing".ProductRequest, "BFT-2 Prod Line" := "THE1_From_BT_To_Mixing".LineProd_Open, "BFT-2 CIP Enable" :=, "BFT-2 CIPLine" :=, "BFT-3 Prod Req" :=, "BFT-3 Prod Line" :=, "BFT-3 CIP Enable" :=, "BFT-3 CIPLine" :=, IN_LDT :=, "CIP Pulse" := "Timer 5S/30s", "CIP Supply ON" :=, "CIP Req OK" :=, "CIP Complete" :=, Out_AV_Header1 =>, Out_AV_Header2 =>, Out_AV_Vinegar =>, Out_AV_Sugar =>, Out_AV_Salt =>, Out_AV_ProWater =>, Out_AV_Homomixer =>, Out_AV_Transfer1 =>, Out_AV_Transfer2 =>, Out_AV_Transfer3 =>, Out_AV_Outlet =>, Out_AV_CIP =>, Out_P_Transfer1 =>, Out_P_Transfer1_Sp =>, Out_P_Transfer2 =>, Out_P_Transfer2_Sp =>, Out_P_Transfer3 =>, Out_P_Transfer3_Sp =>, Out_P_CIP =>, Out_P_CIP_Sp =>, Out_Agi =>, Out_Agi_Sp =>, "Header 1 Req" =>, "Header 2 Req" =>, "Vinegar Req" =>, "Sugar Req" =>, "Salt Req" =>, "ProWater Req" =>, "Homomixer Req" =>, Out_CIP_Req => "Mix_to_CIP".CIP_Request."Blending Cluster 1"."T-21.00_CIP_Request", Out_CIP_Line_Open => "Mix_to_CIP".CIP_Line_OK."Blending Cluster 1"."T-21.00_CIP_LineOK")
   END_RUNG
   RUNG wire#powerrail
      Contact( "Blend_T-20".State."BFT-1 EN" )
   END_RUNG wire#w1
   RUNG wire#powerrail
      Contact( "Blend_T-30".State."BFT-1 EN" )
   END_RUNG wire#w1
   RUNG wire#powerrail
      Contact( "General_Blend".Blend_Cluster1.CIP_Line1."CIP Request" )
   END_RUNG wire#w1
   RUNG wire#powerrail
      Contact( "Blend_T-20".State."BFT-2 EN" )
   END_RUNG wire#w2
   RUNG wire#powerrail
      Contact( "Blend_T-30".State."BFT-2 EN" )
   END_RUNG wire#w2
   RUNG wire#powerrail
      Contact( "General_Blend".Blend_Cluster1.CIP_Line2."CIP Request" )
   END_RUNG wire#w2
   RUNG wire#powerrail
      Contact( "Blend_T-20".State."BFT-3 EN" )
   END_RUNG wire#w3
   RUNG wire#powerrail
      Contact( "Blend_T-30".State."BFT-3 EN" )
   END_RUNG wire#w3
   RUNG wire#powerrail
      Contact( "General_Blend".Blend_Cluster1.CIP_Line3."CIP Request" )
   END_RUNG wire#w3
   RUNG wire#powerrail
      I_Contact( "Blend_T-20"."Header 1 Req" )
      I_Contact( "Blend_T-30"."Header 1 Req" )
      I_Contact( "Blend_T-31"."Header 1 Req" )
      I_Contact( "Blend_T-40"."Header 1 Req" )
      I_Contact( "Blend_T-41"."Header 1 Req" )
      I_Contact( "Preparation to Blend".Header_1_CIP )
   END_RUNG wire#w4
   RUNG wire#powerrail
      I_Contact( "Blend_T-20"."Header 2 Req" )
      I_Contact( "Blend_T-30"."Header 2 Req" )
      I_Contact( "Blend_T-31"."Header 2 Req" )
      I_Contact( "Blend_T-40"."Header 2 Req" )
      I_Contact( "Blend_T-41"."Header 2 Req" )
      I_Contact( "Preparation to Blend".Header_2_CIP )
   END_RUNG wire#w5
   RUNG wire#powerrail
      I_Contact( "Blend_T-20"."Vinegar Req" )
      I_Contact( "Blend_T-30"."Vinegar Req" )
      I_Contact( "Blend_T-31"."Vinegar Req" )
      I_Contact( "Blend_T-40"."Vinegar Req" )
      I_Contact( "Blend_T-41"."Vinegar Req" )
      I_Contact( "T-05_Tomato"."Vinegar Req" )
      I_Contact( "Mix_to_CIP".CIP_Request.Vinegar."T-10.00_CIP_Request" )
   END_RUNG wire#w6
   RUNG wire#powerrail
      I_Contact( "Blend_T-20"."Sugar Req" )
      I_Contact( "Blend_T-30"."Sugar Req" )
      I_Contact( "Blend_T-31"."Sugar Req" )
      I_Contact( "Blend_T-40"."Sugar Req" )
      I_Contact( "Blend_T-41"."Sugar Req" )
   END_RUNG wire#w7
   RUNG wire#powerrail
      I_Contact( "Blend_T-20"."Salt Req" )
      I_Contact( "Blend_T-30"."Salt Req" )
      I_Contact( "Blend_T-31"."Salt Req" )
      I_Contact( "Blend_T-40"."Salt Req" )
      I_Contact( "Blend_T-41"."Salt Req" )
   END_RUNG wire#w8
   RUNG wire#powerrail
      I_Contact( "Blend_T-20"."ProWater Req" )
      I_Contact( "Blend_T-30"."ProWater Req" )
      I_Contact( "Blend_T-31"."ProWater Req" )
      I_Contact( "Blend_T-40"."ProWater Req" )
      I_Contact( "Blend_T-41"."ProWater Req" )
   END_RUNG wire#w9
   RUNG wire#powerrail
      I_Contact( "Blend_T-20"."Homomixer Req" )
      I_Contact( "Mix_to_CIP".CIP_Request.Homomixer."T-12.00_CIP_LineToBlend_Request" )
   END_RUNG wire#w10
   RUNG wire#powerrail
      Contact( "Blend_T-20".Out_CIP_Req )
   END_RUNG wire#w11
   RUNG wire#powerrail
      Contact( "Blend_T-30".Out_CIP_Req )
   END_RUNG wire#w11
   RUNG wire#powerrail
      Contact( "General_Blend".Blend_Cluster1.CIP_Line1."CIP Request" )
   END_RUNG wire#w11
   RUNG wire#powerrail
      Contact( "General_Blend".Blend_Cluster1.CIP_Line2."CIP Request" )
   END_RUNG wire#w11
   RUNG wire#powerrail
      Contact( "General_Blend".Blend_Cluster1.CIP_Line3."CIP Request" )
   END_RUNG wire#w11
   // the same network as SCL:
   "Blend_T-21"(IN_FBAV_Sugar := "Blend_T-21".Out_AV_Sugar,   // "Blend_Tank"
                IN_FBAV_Salt := "Blend_T-21".Out_AV_Salt,
                IN_LT01 := "IO Analog Blending_DB"."LT-21.01".QOUT,
                "BFT-1 Prod Req" := "THE2_From_BT_To_Mixing".ProductRequest,
                "BFT-1 Prod Line" := "THE2_From_BT_To_Mixing".LineProd_Open,
                "BFT-2 Prod Req" := "THE1_From_BT_To_Mixing".ProductRequest,
                "BFT-2 Prod Line" := "THE1_From_BT_To_Mixing".LineProd_Open,
                "Transfer 1 Busy" := "Blend_T-20".State."BFT-1 EN" OR "Blend_T-30".State."BFT-1 EN" OR "General_Blend".Blend_Cluster1.CIP_Line1."CIP Request",
                "Transfer 2 Busy" := "Blend_T-20".State."BFT-2 EN" OR "Blend_T-30".State."BFT-2 EN" OR "General_Blend".Blend_Cluster1.CIP_Line2."CIP Request",
                "Transfer 3 Busy" := "Blend_T-20".State."BFT-3 EN" OR "Blend_T-30".State."BFT-3 EN" OR "General_Blend".Blend_Cluster1.CIP_Line3."CIP Request",
                "Header 1 Available" := NOT "Blend_T-20"."Header 1 Req" AND NOT "Blend_T-30"."Header 1 Req" AND NOT "Blend_T-31"."Header 1 Req" AND NOT "Blend_T-40"."Header 1 Req" AND NOT "Blend_T-41"."Header 1 Req" AND NOT "Preparation to Blend".Header_1_CIP,
                "Header 2 Available" := NOT "Blend_T-20"."Header 2 Req" AND NOT "Blend_T-30"."Header 2 Req" AND NOT "Blend_T-31"."Header 2 Req" AND NOT "Blend_T-40"."Header 2 Req" AND NOT "Blend_T-41"."Header 2 Req" AND NOT "Preparation to Blend".Header_2_CIP,
                "Vinegar Available" := NOT "Blend_T-20"."Vinegar Req" AND NOT "Blend_T-30"."Vinegar Req" AND NOT "Blend_T-31"."Vinegar Req" AND NOT "Blend_T-40"."Vinegar Req" AND NOT "Blend_T-41"."Vinegar Req" AND NOT "T-05_Tomato"."Vinegar Req" AND NOT "Mix_to_CIP".CIP_Request.Vinegar."T-10.00_CIP_Request",
                "Sugar Available" := NOT "Blend_T-20"."Sugar Req" AND NOT "Blend_T-30"."Sugar Req" AND NOT "Blend_T-31"."Sugar Req" AND NOT "Blend_T-40"."Sugar Req" AND NOT "Blend_T-41"."Sugar Req",
                "Salt Available" := NOT "Blend_T-20"."Salt Req" AND NOT "Blend_T-30"."Salt Req" AND NOT "Blend_T-31"."Salt Req" AND NOT "Blend_T-40"."Salt Req" AND NOT "Blend_T-41"."Salt Req",
                "ProWater Available" := NOT "Blend_T-20"."ProWater Req" AND NOT "Blend_T-30"."ProWater Req" AND NOT "Blend_T-31"."ProWater Req" AND NOT "Blend_T-40"."ProWater Req" AND NOT "Blend_T-41"."ProWater Req",
                "Homomixer Available" := NOT "Blend_T-20"."Homomixer Req" AND NOT "Mix_to_CIP".CIP_Request.Homomixer."T-12.00_CIP_LineToBlend_Request",
                "CIP Pulse" := "Timer 5S/30s",
                "CIP Busy" := "Blend_T-20".Out_CIP_Req OR "Blend_T-30".Out_CIP_Req OR "General_Blend".Blend_Cluster1.CIP_Line1."CIP Request" OR "General_Blend".Blend_Cluster1.CIP_Line2."CIP Request" OR "General_Blend".Blend_Cluster1.CIP_Line3."CIP Request",
                Out_CIP_Req => "Mix_to_CIP".CIP_Request."Blending Cluster 1"."T-21.00_CIP_Request",
                Out_CIP_Line_Open => "Mix_to_CIP".CIP_Line_OK."Blending Cluster 1"."T-21.00_CIP_LineOK");
END_REGION

REGION Network 40: Blending T-21 Feedback Valve
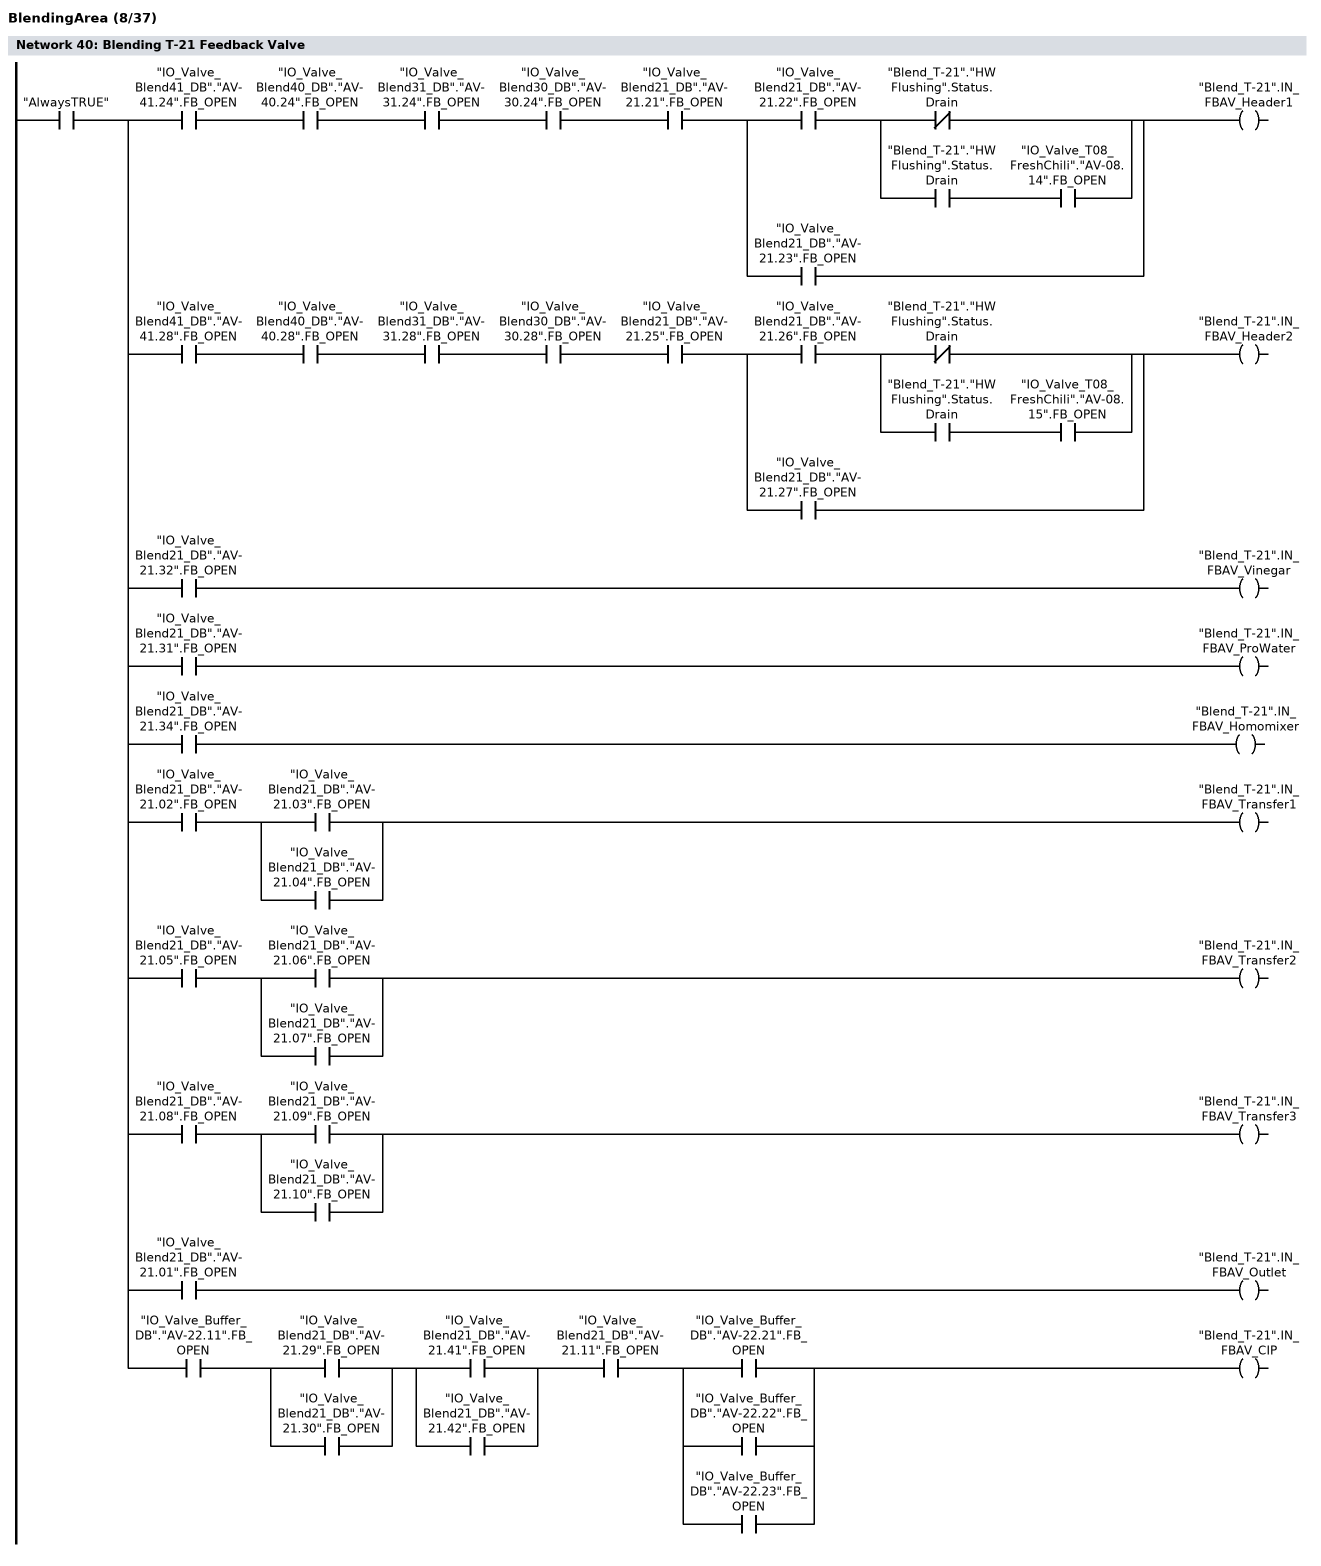
   RUNG wire#powerrail
      Contact( "AlwaysTRUE" )
      wire#w1
      Contact( "IO_Valve_Blend41_DB"."AV-41.24".FB_OPEN )
      Contact( "IO_Valve_Blend40_DB"."AV-40.24".FB_OPEN )
      Contact( "IO_Valve_Blend31_DB"."AV-31.24".FB_OPEN )
      Contact( "IO_Valve_Blend30_DB"."AV-30.24".FB_OPEN )
      Contact( "IO_Valve_Blend21_DB"."AV-21.21".FB_OPEN )
      wire#w2
      Contact( "IO_Valve_Blend21_DB"."AV-21.22".FB_OPEN )
      wire#w3
      I_Contact( "Blend_T-21"."HW Flushing".Status.Drain )
      wire#w4
      Coil( "Blend_T-21".IN_FBAV_Header1 )
   END_RUNG
   RUNG wire#w3
      Contact( "Blend_T-21"."HW Flushing".Status.Drain )
      Contact( "IO_Valve_T08_FreshChili"."AV-08.14".FB_OPEN )
   END_RUNG wire#w4
   RUNG wire#w2
      Contact( "IO_Valve_Blend21_DB"."AV-21.23".FB_OPEN )
   END_RUNG wire#w4
   RUNG wire#w1
      Contact( "IO_Valve_Blend41_DB"."AV-41.28".FB_OPEN )
      Contact( "IO_Valve_Blend40_DB"."AV-40.28".FB_OPEN )
      Contact( "IO_Valve_Blend31_DB"."AV-31.28".FB_OPEN )
      Contact( "IO_Valve_Blend30_DB"."AV-30.28".FB_OPEN )
      Contact( "IO_Valve_Blend21_DB"."AV-21.25".FB_OPEN )
      wire#w5
      Contact( "IO_Valve_Blend21_DB"."AV-21.26".FB_OPEN )
      wire#w6
      I_Contact( "Blend_T-21"."HW Flushing".Status.Drain )
      wire#w7
      Coil( "Blend_T-21".IN_FBAV_Header2 )
   END_RUNG
   RUNG wire#w6
      Contact( "Blend_T-21"."HW Flushing".Status.Drain )
      Contact( "IO_Valve_T08_FreshChili"."AV-08.15".FB_OPEN )
   END_RUNG wire#w7
   RUNG wire#w5
      Contact( "IO_Valve_Blend21_DB"."AV-21.27".FB_OPEN )
   END_RUNG wire#w7
   RUNG wire#w1
      Contact( "IO_Valve_Blend21_DB"."AV-21.32".FB_OPEN )
      Coil( "Blend_T-21".IN_FBAV_Vinegar )
   END_RUNG
   RUNG wire#w1
      Contact( "IO_Valve_Blend21_DB"."AV-21.31".FB_OPEN )
      Coil( "Blend_T-21".IN_FBAV_ProWater )
   END_RUNG
   RUNG wire#w1
      Contact( "IO_Valve_Blend21_DB"."AV-21.34".FB_OPEN )
      Coil( "Blend_T-21".IN_FBAV_Homomixer )
   END_RUNG
   RUNG wire#w1
      Contact( "IO_Valve_Blend21_DB"."AV-21.02".FB_OPEN )
      wire#w8
      Contact( "IO_Valve_Blend21_DB"."AV-21.03".FB_OPEN )
      wire#w9
      Coil( "Blend_T-21".IN_FBAV_Transfer1 )
   END_RUNG
   RUNG wire#w8
      Contact( "IO_Valve_Blend21_DB"."AV-21.04".FB_OPEN )
   END_RUNG wire#w9
   RUNG wire#w1
      Contact( "IO_Valve_Blend21_DB"."AV-21.05".FB_OPEN )
      wire#w10
      Contact( "IO_Valve_Blend21_DB"."AV-21.06".FB_OPEN )
      wire#w11
      Coil( "Blend_T-21".IN_FBAV_Transfer2 )
   END_RUNG
   RUNG wire#w10
      Contact( "IO_Valve_Blend21_DB"."AV-21.07".FB_OPEN )
   END_RUNG wire#w11
   RUNG wire#w1
      Contact( "IO_Valve_Blend21_DB"."AV-21.08".FB_OPEN )
      wire#w12
      Contact( "IO_Valve_Blend21_DB"."AV-21.09".FB_OPEN )
      wire#w13
      Coil( "Blend_T-21".IN_FBAV_Transfer3 )
   END_RUNG
   RUNG wire#w12
      Contact( "IO_Valve_Blend21_DB"."AV-21.10".FB_OPEN )
   END_RUNG wire#w13
   RUNG wire#w1
      Contact( "IO_Valve_Blend21_DB"."AV-21.01".FB_OPEN )
      Coil( "Blend_T-21".IN_FBAV_Outlet )
   END_RUNG
   RUNG wire#w1
      Contact( "IO_Valve_Buffer_DB"."AV-22.11".FB_OPEN )
      wire#w14
      Contact( "IO_Valve_Blend21_DB"."AV-21.29".FB_OPEN )
      wire#w15
      Contact( "IO_Valve_Blend21_DB"."AV-21.41".FB_OPEN )
      wire#w16
      Contact( "IO_Valve_Blend21_DB"."AV-21.11".FB_OPEN )
      wire#w17
      Contact( "IO_Valve_Buffer_DB"."AV-22.21".FB_OPEN )
      wire#w18
      Coil( "Blend_T-21".IN_FBAV_CIP )
   END_RUNG
   RUNG wire#w14
      Contact( "IO_Valve_Blend21_DB"."AV-21.30".FB_OPEN )
   END_RUNG wire#w15
   RUNG wire#w15
      Contact( "IO_Valve_Blend21_DB"."AV-21.42".FB_OPEN )
   END_RUNG wire#w16
   RUNG wire#w17
      Contact( "IO_Valve_Buffer_DB"."AV-22.22".FB_OPEN )
   END_RUNG wire#w18
   RUNG wire#w17
      Contact( "IO_Valve_Buffer_DB"."AV-22.23".FB_OPEN )
   END_RUNG wire#w18
   // the same network as SCL:
   "Blend_T-21".IN_FBAV_Header1 := "AlwaysTRUE" AND "IO_Valve_Blend41_DB"."AV-41.24".FB_OPEN AND "IO_Valve_Blend40_DB"."AV-40.24".FB_OPEN AND "IO_Valve_Blend31_DB"."AV-31.24".FB_OPEN AND "IO_Valve_Blend30_DB"."AV-30.24".FB_OPEN AND "IO_Valve_Blend21_DB"."AV-21.21".FB_OPEN AND (("IO_Valve_Blend21_DB"."AV-21.22".FB_OPEN AND (NOT "Blend_T-21"."HW Flushing".Status.Drain OR ("Blend_T-21"."HW Flushing".Status.Drain AND "IO_Valve_T08_FreshChili"."AV-08.14".FB_OPEN))) OR "IO_Valve_Blend21_DB"."AV-21.23".FB_OPEN);
   "Blend_T-21".IN_FBAV_Header2 := "AlwaysTRUE" AND "IO_Valve_Blend41_DB"."AV-41.28".FB_OPEN AND "IO_Valve_Blend40_DB"."AV-40.28".FB_OPEN AND "IO_Valve_Blend31_DB"."AV-31.28".FB_OPEN AND "IO_Valve_Blend30_DB"."AV-30.28".FB_OPEN AND "IO_Valve_Blend21_DB"."AV-21.25".FB_OPEN AND (("IO_Valve_Blend21_DB"."AV-21.26".FB_OPEN AND (NOT "Blend_T-21"."HW Flushing".Status.Drain OR ("Blend_T-21"."HW Flushing".Status.Drain AND "IO_Valve_T08_FreshChili"."AV-08.15".FB_OPEN))) OR "IO_Valve_Blend21_DB"."AV-21.27".FB_OPEN);
   "Blend_T-21".IN_FBAV_Vinegar := "AlwaysTRUE" AND "IO_Valve_Blend21_DB"."AV-21.32".FB_OPEN;
   "Blend_T-21".IN_FBAV_ProWater := "AlwaysTRUE" AND "IO_Valve_Blend21_DB"."AV-21.31".FB_OPEN;
   "Blend_T-21".IN_FBAV_Homomixer := "AlwaysTRUE" AND "IO_Valve_Blend21_DB"."AV-21.34".FB_OPEN;
   "Blend_T-21".IN_FBAV_Transfer1 := "AlwaysTRUE" AND "IO_Valve_Blend21_DB"."AV-21.02".FB_OPEN AND ("IO_Valve_Blend21_DB"."AV-21.03".FB_OPEN OR "IO_Valve_Blend21_DB"."AV-21.04".FB_OPEN);
   "Blend_T-21".IN_FBAV_Transfer2 := "AlwaysTRUE" AND "IO_Valve_Blend21_DB"."AV-21.05".FB_OPEN AND ("IO_Valve_Blend21_DB"."AV-21.06".FB_OPEN OR "IO_Valve_Blend21_DB"."AV-21.07".FB_OPEN);
   "Blend_T-21".IN_FBAV_Transfer3 := "AlwaysTRUE" AND "IO_Valve_Blend21_DB"."AV-21.08".FB_OPEN AND ("IO_Valve_Blend21_DB"."AV-21.09".FB_OPEN OR "IO_Valve_Blend21_DB"."AV-21.10".FB_OPEN);
   "Blend_T-21".IN_FBAV_Outlet := "AlwaysTRUE" AND "IO_Valve_Blend21_DB"."AV-21.01".FB_OPEN;
   "Blend_T-21".IN_FBAV_CIP := "AlwaysTRUE" AND "IO_Valve_Buffer_DB"."AV-22.11".FB_OPEN AND ("IO_Valve_Blend21_DB"."AV-21.29".FB_OPEN OR "IO_Valve_Blend21_DB"."AV-21.30".FB_OPEN) AND ("IO_Valve_Blend21_DB"."AV-21.41".FB_OPEN OR "IO_Valve_Blend21_DB"."AV-21.42".FB_OPEN) AND "IO_Valve_Blend21_DB"."AV-21.11".FB_OPEN AND ("IO_Valve_Buffer_DB"."AV-22.21".FB_OPEN OR "IO_Valve_Buffer_DB"."AV-22.22".FB_OPEN OR "IO_Valve_Buffer_DB"."AV-22.23".FB_OPEN);
END_REGION

REGION Network 41: Blending T-21 Feedback Pump
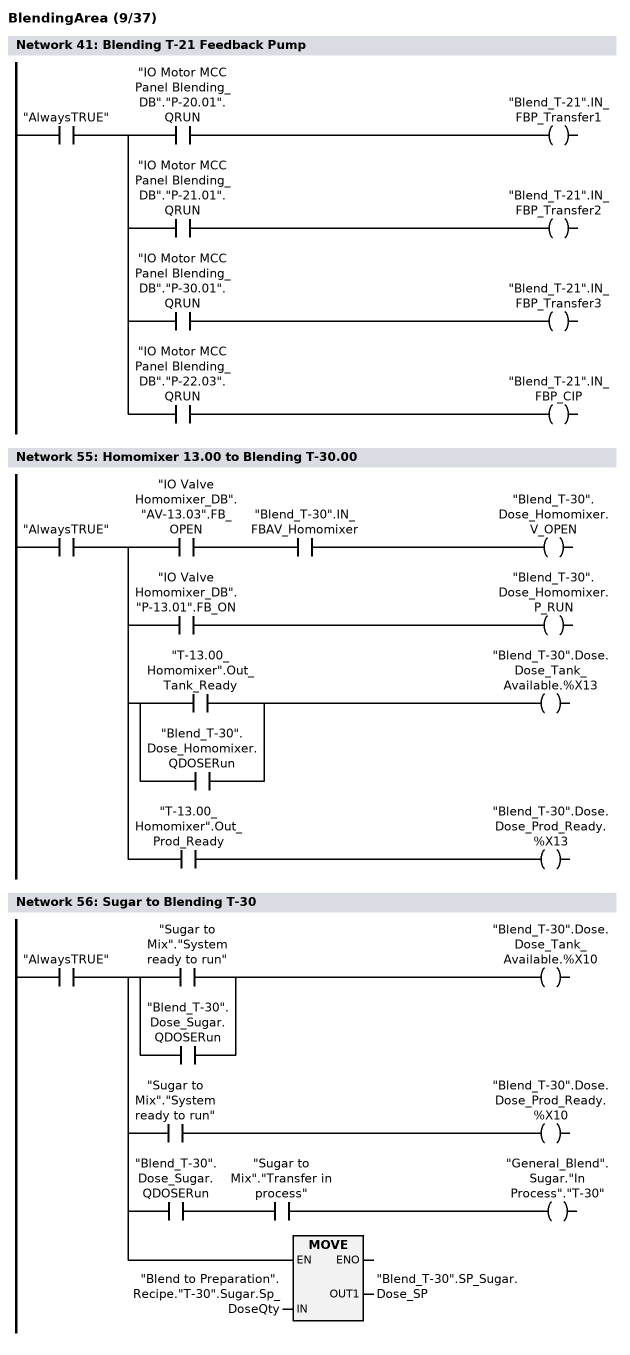
   RUNG wire#powerrail
      Contact( "AlwaysTRUE" )
      wire#w1
      Contact( "IO Motor MCC Panel Blending_DB"."P-20.01".QRUN )
      Coil( "Blend_T-21".IN_FBP_Transfer1 )
   END_RUNG
   RUNG wire#w1
      Contact( "IO Motor MCC Panel Blending_DB"."P-21.01".QRUN )
      Coil( "Blend_T-21".IN_FBP_Transfer2 )
   END_RUNG
   RUNG wire#w1
      Contact( "IO Motor MCC Panel Blending_DB"."P-30.01".QRUN )
      Coil( "Blend_T-21".IN_FBP_Transfer3 )
   END_RUNG
   RUNG wire#w1
      Contact( "IO Motor MCC Panel Blending_DB"."P-22.03".QRUN )
      Coil( "Blend_T-21".IN_FBP_CIP )
   END_RUNG
   // the same network as SCL:
   "Blend_T-21".IN_FBP_Transfer1 := "AlwaysTRUE" AND "IO Motor MCC Panel Blending_DB"."P-20.01".QRUN;
   "Blend_T-21".IN_FBP_Transfer2 := "AlwaysTRUE" AND "IO Motor MCC Panel Blending_DB"."P-21.01".QRUN;
   "Blend_T-21".IN_FBP_Transfer3 := "AlwaysTRUE" AND "IO Motor MCC Panel Blending_DB"."P-30.01".QRUN;
   "Blend_T-21".IN_FBP_CIP := "AlwaysTRUE" AND "IO Motor MCC Panel Blending_DB"."P-22.03".QRUN;
END_REGION

NETWORK
TITLE = Blending T-21 to Preparation
//to ChiliAwetan1
      O     "Blend_T-21".Dose_ChiliAwetan1.QDOSERun;  //Dose Run
      =     "Blend to Preparation"."T-21".Raw_Material.ChiliAwetan_1.DoseRun;
      O     "Blend_T-21".Dose_ChiliAwetan1.QHELD;  //Dose Held
      =     "Blend to Preparation"."T-21".Raw_Material.ChiliAwetan_1.DoseHeld;
      O     "Blend_T-21".Dose_ChiliAwetan1.QDoseComplete;  //Dose Complete
      =     "Blend to Preparation"."T-21".Raw_Material.ChiliAwetan_1.DoseComplete;
      O     "Blend_T-21".Dose_ChiliAwetan1.V_CMD;  //Valve Command
      =     "Blend to Preparation"."T-21".Raw_Material.ChiliAwetan_1.ValveCMD;
      O     "Blend_T-21".Dose_ChiliAwetan1.P_CMD;  //Pump Command
      =     "Blend to Preparation"."T-21".Raw_Material.ChiliAwetan_1.PumpCMD;
      O     "Blend_T-21".Dose.Dose_Header_Req.%X0;  //Header 1 Req
      =     "Blend to Preparation"."T-21".Raw_Material.ChiliAwetan_1.Header1_Req;
      O     "Blend_T-21".Dose.Dose_Header_Req.%X16;  //Header 2 Req
      =     "Blend to Preparation"."T-21".Raw_Material.ChiliAwetan_1.Header2_Req;
      L     "Blend to Preparation".Recipe."T-21".ChiliAwetan_1.Sp_DoseQty;  //Load Sp Dose From Recipe
      T     "Blend_T-21".SP_ChiliAwetan1.Dose_SP;
      L     "Blend_T-21".Dose_ChiliAwetan1.P_SPEED;  //Pump Speed
      T     "Blend to Preparation".Recipe."T-21".ChiliAwetan_1.SP_PumpSpeed;

//to ChiliAwetan2
      O     "Blend_T-21".Dose_ChiliAwetan2.QDOSERun;  //Dose Run
      =     "Blend to Preparation"."T-21".Raw_Material.ChiliAwetan_2.DoseRun;
      O     "Blend_T-21".Dose_ChiliAwetan2.QHELD;  //Dose Held
      =     "Blend to Preparation"."T-21".Raw_Material.ChiliAwetan_2.DoseHeld;
      O     "Blend_T-21".Dose_ChiliAwetan2.QDoseComplete;  //Dose Complete
      =     "Blend to Preparation"."T-21".Raw_Material.ChiliAwetan_2.DoseComplete;
      O     "Blend_T-21".Dose_ChiliAwetan2.V_CMD;  //Valve Command
      =     "Blend to Preparation"."T-21".Raw_Material.ChiliAwetan_2.ValveCMD;
      O     "Blend_T-21".Dose_ChiliAwetan2.P_CMD;  //Pump Command
      =     "Blend to Preparation"."T-21".Raw_Material.ChiliAwetan_2.PumpCMD;
      O     "Blend_T-21".Dose.Dose_Header_Req.%X1;  //Header 1 Req
      =     "Blend to Preparation"."T-21".Raw_Material.ChiliAwetan_2.Header1_Req;
      O     "Blend_T-21".Dose.Dose_Header_Req.%X17;  //Header 2 Req
      =     "Blend to Preparation"."T-21".Raw_Material.ChiliAwetan_2.Header2_Req;
      L     "Blend to Preparation".Recipe."T-21".ChiliAwetan_2.Sp_DoseQty;  //Load Sp Dose From Recipe
      T     "Blend_T-21".SP_ChiliAwetan2.Dose_SP;
      L     "Blend_T-21".Dose_ChiliAwetan2.P_SPEED;  //Pump Speed
      T     "Blend to Preparation".Recipe."T-21".ChiliAwetan_2.SP_PumpSpeed;

//to ChiliAwetan3
      O     "Blend_T-21".Dose_ChiliAwetan3.QDOSERun;  //Dose Run
      =     "Blend to Preparation"."T-21".Raw_Material.ChiliAwetan_3.DoseRun;
      O     "Blend_T-21".Dose_ChiliAwetan3.QHELD;  //Dose Held
      =     "Blend to Preparation"."T-21".Raw_Material.ChiliAwetan_3.DoseHeld;
      O     "Blend_T-21".Dose_ChiliAwetan3.QDoseComplete;  //Dose Complete
      =     "Blend to Preparation"."T-21".Raw_Material.ChiliAwetan_3.DoseComplete;
      O     "Blend_T-21".Dose_ChiliAwetan3.V_CMD;  //Valve Command
      =     "Blend to Preparation"."T-21".Raw_Material.ChiliAwetan_3.ValveCMD;
      O     "Blend_T-21".Dose_ChiliAwetan3.P_CMD;  //Pump Command
      =     "Blend to Preparation"."T-21".Raw_Material.ChiliAwetan_3.PumpCMD;
      O     "Blend_T-21".Dose.Dose_Header_Req.%X2;  //Header 1 Req
      =     "Blend to Preparation"."T-21".Raw_Material.ChiliAwetan_3.Header1_Req;
      O     "Blend_T-21".Dose.Dose_Header_Req.%X18;  //Header 2 Req
      =     "Blend to Preparation"."T-21".Raw_Material.ChiliAwetan_3.Header2_Req;
      L     "Blend to Preparation".Recipe."T-21".ChiliAwetan_3.Sp_DoseQty;  //Load Sp Dose From Recipe
      T     "Blend_T-21".SP_ChiliAwetan3.Dose_SP;
      L     "Blend_T-21".Dose_ChiliAwetan3.P_SPEED;  //Pump Speed
      T     "Blend to Preparation".Recipe."T-21".ChiliAwetan_3.SP_PumpSpeed;

//to Tomato
      O     "Blend_T-21".Dose_Tomato.QDOSERun;  //Dose Run
      =     "Blend to Preparation"."T-21".Raw_Material.Tomato.DoseRun;
      O     "Blend_T-21".Dose_Tomato.QHELD;  //Dose Held
      =     "Blend to Preparation"."T-21".Raw_Material.Tomato.DoseHeld;
      O     "Blend_T-21".Dose_Tomato.QDoseComplete;  //Dose Complete
      =     "Blend to Preparation"."T-21".Raw_Material.Tomato.DoseComplete;
      O     "Blend_T-21".Dose_Tomato.V_CMD;  //Valve Command
      =     "Blend to Preparation"."T-21".Raw_Material.Tomato.ValveCMD;
      O     "Blend_T-21".Dose_Tomato.P_CMD;  //Pump Command
      =     "Blend to Preparation"."T-21".Raw_Material.Tomato.PumpCMD;
      O     "Blend_T-21".Dose.Dose_Header_Req.%X3;  //Header 1 Req
      =     "Blend to Preparation"."T-21".Raw_Material.Tomato.Header1_Req;
      O     "Blend_T-21".Dose.Dose_Header_Req.%X19;  //Header 2 Req
      =     "Blend to Preparation"."T-21".Raw_Material.Tomato.Header2_Req;
      L     "Blend to Preparation".Recipe."T-21".Tomato.Sp_DoseQty;  //Load Sp Dose From Recipe
      T     "Blend_T-21".SP_Tomato.Dose_SP;
      L     "Blend_T-21".Dose_Tomato.P_SPEED;  //Pump Speed
      T     "Blend to Preparation".Recipe."T-21".Tomato.SP_PumpSpeed;

//to ChiliFresh1
      O     "Blend_T-21".Dose_ChiliFresh1.QDOSERun;  //Dose Run
      =     "Blend to Preparation"."T-21".Raw_Material.ChiliFresh_1.DoseRun;
      O     "Blend_T-21".Dose_ChiliFresh1.QHELD;  //Dose Held
      =     "Blend to Preparation"."T-21".Raw_Material.ChiliFresh_1.DoseHeld;
      O     "Blend_T-21".Dose_ChiliFresh1.QDoseComplete;  //Dose Complete
      =     "Blend to Preparation"."T-21".Raw_Material.ChiliFresh_1.DoseComplete;
      O     "Blend_T-21".Dose_ChiliFresh1.V_CMD;  //Valve Command
      =     "Blend to Preparation"."T-21".Raw_Material.ChiliFresh_1.ValveCMD;
      O     "Blend_T-21".Dose_ChiliFresh1.P_CMD;  //Pump Command
      =     "Blend to Preparation"."T-21".Raw_Material.ChiliFresh_1.PumpCMD;
      O     "Blend_T-21".Dose.Dose_Header_Req.%X4;  //Header 1 Req
      =     "Blend to Preparation"."T-21".Raw_Material.ChiliFresh_1.Header1_Req;
      O     "Blend_T-21".Dose.Dose_Header_Req.%X20;  //Header 2 Req
      =     "Blend to Preparation"."T-21".Raw_Material.ChiliFresh_1.Header2_Req;
      L     "Blend to Preparation".Recipe."T-21".ChiliFresh_1.Sp_DoseQty;  //Load Sp Dose From Recipe
      T     "Blend_T-21".SP_ChiliFresh1.Dose_SP;
      L     "Blend_T-21".Dose_ChiliFresh1.P_SPEED;  //Pump Speed
      T     "Blend to Preparation".Recipe."T-21".ChiliFresh_1.SP_PumpSpeed;

//to ChiliFresh2
      O     "Blend_T-21".Dose_ChiliFresh2.QDOSERun;  //Dose Run
      =     "Blend to Preparation"."T-21".Raw_Material.ChiliFresh_2.DoseRun;
      O     "Blend_T-21".Dose_ChiliFresh2.QHELD;  //Dose Held
      =     "Blend to Preparation"."T-21".Raw_Material.ChiliFresh_2.DoseHeld;
      O     "Blend_T-21".Dose_ChiliFresh2.QDoseComplete;  //Dose Complete
      =     "Blend to Preparation"."T-21".Raw_Material.ChiliFresh_2.DoseComplete;
      O     "Blend_T-21".Dose_ChiliFresh2.V_CMD;  //Valve Command
      =     "Blend to Preparation"."T-21".Raw_Material.ChiliFresh_2.ValveCMD;
      O     "Blend_T-21".Dose_ChiliFresh2.P_CMD;  //Pump Command
      =     "Blend to Preparation"."T-21".Raw_Material.ChiliFresh_2.PumpCMD;
      O     "Blend_T-21".Dose.Dose_Header_Req.%X5;  //Header 1 Req
      =     "Blend to Preparation"."T-21".Raw_Material.ChiliFresh_2.Header1_Req;
      O     "Blend_T-21".Dose.Dose_Header_Req.%X21;  //Header 2 Req
      =     "Blend to Preparation"."T-21".Raw_Material.ChiliFresh_2.Header2_Req;
      L     "Blend to Preparation".Recipe."T-21".ChiliFresh_2.Sp_DoseQty;  //Load Sp Dose From Recipe
      T     "Blend_T-21".SP_ChiliFresh2.Dose_SP;
      L     "Blend_T-21".Dose_ChiliFresh2.P_SPEED;  //Pump Speed
      T     "Blend to Preparation".Recipe."T-21".ChiliFresh_2.SP_PumpSpeed;

//to ChiliFresh3
      O     "Blend_T-21".Dose_ChiliFresh3.QDOSERun;  //Dose Run
      =     "Blend to Preparation"."T-21".Raw_Material.ChiliFresh_3.DoseRun;
      O     "Blend_T-21".Dose_ChiliFresh3.QHELD;  //Dose Held
      =     "Blend to Preparation"."T-21".Raw_Material.ChiliFresh_3.DoseHeld;
      O     "Blend_T-21".Dose_ChiliFresh3.QDoseComplete;  //Dose Complete
      =     "Blend to Preparation"."T-21".Raw_Material.ChiliFresh_3.DoseComplete;
      O     "Blend_T-21".Dose_ChiliFresh3.V_CMD;  //Valve Command
      =     "Blend to Preparation"."T-21".Raw_Material.ChiliFresh_3.ValveCMD;
      O     "Blend_T-21".Dose_ChiliFresh3.P_CMD;  //Pump Command
      =     "Blend to Preparation"."T-21".Raw_Material.ChiliFresh_3.PumpCMD;
      O     "Blend_T-21".Dose.Dose_Header_Req.%X6;  //Header 1 Req
      =     "Blend to Preparation"."T-21".Raw_Material.ChiliFresh_3.Header1_Req;
      O     "Blend_T-21".Dose.Dose_Header_Req.%X22;  //Header 2 Req
      =     "Blend to Preparation"."T-21".Raw_Material.ChiliFresh_3.Header2_Req;
      L     "Blend to Preparation".Recipe."T-21".ChiliFresh_3.Sp_DoseQty;  //Load Sp Dose From Recipe
      T     "Blend_T-21".SP_ChiliFresh3.Dose_SP;
      L     "Blend_T-21".Dose_ChiliFresh3.P_SPEED;  //Pump Speed
      T     "Blend to Preparation".Recipe."T-21".ChiliFresh_3.SP_PumpSpeed;

//to Garlic
      O     "Blend_T-21".Dose_Garlic.QDOSERun;  //Dose Run
      =     "Blend to Preparation"."T-21".Raw_Material.Garlic.DoseRun;
      O     "Blend_T-21".Dose_Garlic.QHELD;  //Dose Held
      =     "Blend to Preparation"."T-21".Raw_Material.Garlic.DoseHeld;
      O     "Blend_T-21".Dose_Garlic.QDoseComplete;  //Dose Complete
      =     "Blend to Preparation"."T-21".Raw_Material.Garlic.DoseComplete;
      O     "Blend_T-21".Dose_Garlic.V_CMD;  //Valve Command
      =     "Blend to Preparation"."T-21".Raw_Material.Garlic.ValveCMD;
      O     "Blend_T-21".Dose_Garlic.P_CMD;  //Pump Command
      =     "Blend to Preparation"."T-21".Raw_Material.Garlic.PumpCMD;
      O     "Blend_T-21".Dose.Dose_Header_Req.%X7;  //Header 1 Req
      =     "Blend to Preparation"."T-21".Raw_Material.Garlic.Header1_Req;
      O     "Blend_T-21".Dose.Dose_Header_Req.%X23;  //Header 2 Req
      =     "Blend to Preparation"."T-21".Raw_Material.Garlic.Header2_Req;
      L     "Blend to Preparation".Recipe."T-21".Garlic.Sp_DoseQty;  //Load Sp Dose From Recipe
      T     "Blend_T-21".SP_Garlic.Dose_SP;
      L     "Blend_T-21".Dose_Garlic.P_SPEED;  //Pump Speed
      T     "Blend to Preparation".Recipe."T-21".Garlic.SP_PumpSpeed;

//to Vinegar
      O     "Blend_T-21".Dose_Vinegar.QDOSERun;  //Dose Run
      =     "Blend to Preparation"."T-21".Raw_Material.Vinegar.DoseRun;
      O     "Blend_T-21".Dose_Vinegar.QHELD;  //Dose Held
      =     "Blend to Preparation"."T-21".Raw_Material.Vinegar.DoseHeld;
      O     "Blend_T-21".Dose_Vinegar.QDoseComplete;  //Dose Complete
      =     "Blend to Preparation"."T-21".Raw_Material.Vinegar.DoseComplete;
      O     "Blend_T-21".Dose_Vinegar.V_CMD;  //Valve Command
      =     "Blend to Preparation"."T-21".Raw_Material.Vinegar.ValveCMD;
      O     "Blend_T-21".Dose_Vinegar.P_CMD;  //Pump Command
      =     "Blend to Preparation"."T-21".Raw_Material.Vinegar.PumpCMD;
      L     "Blend to Preparation".Recipe."T-21".Vinegar.Sp_DoseQty;  //Load Sp Dose From Recipe
      T     "Blend_T-21".SP_Vinegar.Dose_SP;
      L     "Blend_T-21".Dose_Vinegar.P_SPEED;  //Pump Speed
      T     "Blend to Preparation".Recipe."T-21".Vinegar.SP_PumpSpeed;

//to HW
      O     "Blend_T-21".Dose_HW.QDOSERun;  //Dose Run
      =     "Blend to Preparation"."T-21".Raw_Material.HW.DoseRun;
      O     "Blend_T-21".Dose_HW.QHELD;  //Dose Held
      =     "Blend to Preparation"."T-21".Raw_Material.HW.DoseHeld;
      O     "Blend_T-21".Dose_HW.QDoseComplete;  //Dose Complete
      =     "Blend to Preparation"."T-21".Raw_Material.HW.DoseComplete;
      O     "Blend_T-21".Dose_HW.V_CMD;  //Valve Command
      =     "Blend to Preparation"."T-21".Raw_Material.HW.ValveCMD;
      O     "Blend_T-21".Dose_HW.P_CMD;  //Pump Command
      =     "Blend to Preparation"."T-21".Raw_Material.HW.PumpCMD;
      O     "Blend_T-21".Dose.Dose_Header_Req.%X8;  //Header 1 Req
      =     "Blend to Preparation"."T-21".Raw_Material.HW.Header1_Req;
      O     "Blend_T-21".Dose.Dose_Header_Req.%X24;  //Header 2 Req
      =     "Blend to Preparation"."T-21".Raw_Material.HW.Header2_Req;

      L     "Blend to Preparation".Recipe."T-21".HW.Sp_Flush_to_BlendQty;  //Load Flush to Blend Sp Dose From Recipe
      T     "Blend_T-21"."HW Flushing".Qty."Flush to Blend Qty";
      L     "Blend to Preparation".Recipe."T-21".HW.Sp_Flush_to_DrainQty;  //Load Flush to Blend Sp Dose From Recipe
      T     "Blend_T-21"."HW Flushing".Qty."Flush to Drain Qty";  //Load Drain Time from recipe
      L     "Blend to Preparation".Recipe."T-21".HW.Sp_DrainTime;
      T     "Blend_T-21"."HW Flushing".TimeDrain_SP;

      L     "Blend_T-21".Dose_HW.P_SPEED;  //Pump Speed
      T     "Blend to Preparation".Recipe."T-21".HW.SP_PumpSpeed;


//General
      O     "Blend_T-21".IN_FBAV_Header1;
      =     "Blend to Preparation"."T-21".LineHeader1_OK;
      O     "Blend_T-21".IN_FBAV_Header2;
      =     "Blend to Preparation"."T-21".LineHeader2_OK;
      O     "Blend_T-21".IN_FBAV_Vinegar;
      =     "Blend to Preparation"."T-21".LineVinegar_OK;


NETWORK
TITLE = ChiliAwetan1 to Blending T-30
//Valve Open
      A     "Preparation to Blend"."T-02_ChiliAwetan_1".Valve_Open;
      A(;
      O(;
      A     "Blend_T-30".Dose.Dose_Header_Req.%X0;
      A     "Blend_T-30".IN_FBAV_Header1;
      );
      O(;
      A     "Blend_T-30".Dose.Dose_Header_Req.%X16;
      A     "Blend_T-30".IN_FBAV_Header2;
      );
      );
      =     "Blend_T-30".Dose_ChiliAwetan1.V_OPEN;
//Pump On
      O     "Preparation to Blend"."T-02_ChiliAwetan_1".Pump_Run;
      =     "Blend_T-30".Dose_ChiliAwetan1.P_RUN;
//Tank Available
      O     "Preparation to Blend"."T-02_ChiliAwetan_1".Tank_Available;
      O     "Blend_T-30".Dose_ChiliAwetan1.QDOSERun;
      =     "Blend_T-30".Dose.Dose_Tank_Available.%X0;
//Product Ready
      O     "Preparation to Blend"."T-02_ChiliAwetan_1".Product_Ready;
      =     "Blend_T-30".Dose.Dose_Prod_Ready.%X0;
//Level Tank
      L     "Preparation to Blend"."T-02_ChiliAwetan_1".Level;
      T     "Blend_T-30"."Dose_Level_%"."ChiliAwetan1%";


NETWORK
TITLE = ChiliAwetan2 to Blending T-30
//Valve Open
      A     "Preparation to Blend"."T-03_ChiliAwetan_2".Valve_Open;
      A(;
      O(;
      A     "Blend_T-30".Dose.Dose_Header_Req.%X1;
      A     "Blend_T-30".IN_FBAV_Header1;
      );
      O(;
      A     "Blend_T-30".Dose.Dose_Header_Req.%X17;
      A     "Blend_T-30".IN_FBAV_Header2;
      );
      );
      =     "Blend_T-30".Dose_ChiliAwetan2.V_OPEN;
//Pump On
      O     "Preparation to Blend"."T-03_ChiliAwetan_2".Pump_Run;
      =     "Blend_T-30".Dose_ChiliAwetan2.P_RUN;
//Tank Available
      O     "Preparation to Blend"."T-03_ChiliAwetan_2".Tank_Available;
      O     "Blend_T-30".Dose_ChiliAwetan2.QDOSERun;
      =     "Blend_T-30".Dose.Dose_Tank_Available.%X1;
//Product Ready
      O     "Preparation to Blend"."T-03_ChiliAwetan_2".Product_Ready;
      =     "Blend_T-30".Dose.Dose_Prod_Ready.%X1;
//Level Tank
      L     "Preparation to Blend"."T-03_ChiliAwetan_2".Level;
      T     "Blend_T-30"."Dose_Level_%"."ChiliAwetan2%";


NETWORK
TITLE = ChiliAwetan3 to Blending T-30
//Valve Open
      A     "Preparation to Blend"."T-04_ChiliAwetan_3".Valve_Open;
      A(;
      O(;
      A     "Blend_T-30".Dose.Dose_Header_Req.%X2;
      A     "Blend_T-30".IN_FBAV_Header1;
      );
      O(;
      A     "Blend_T-30".Dose.Dose_Header_Req.%X18;
      A     "Blend_T-30".IN_FBAV_Header2;
      );
      );
      =     "Blend_T-30".Dose_ChiliAwetan3.V_OPEN;
//Pump On
      O     "Preparation to Blend"."T-04_ChiliAwetan_3".Pump_Run;
      =     "Blend_T-30".Dose_ChiliAwetan3.P_RUN;
//Tank Available
      O     "Preparation to Blend"."T-04_ChiliAwetan_3".Tank_Available;
      O     "Blend_T-30".Dose_ChiliAwetan3.QDOSERun;
      =     "Blend_T-30".Dose.Dose_Tank_Available.%X2;
//Product Ready
      O     "Preparation to Blend"."T-04_ChiliAwetan_3".Product_Ready;
      =     "Blend_T-30".Dose.Dose_Prod_Ready.%X2;
//Level Tank
      L     "Preparation to Blend"."T-04_ChiliAwetan_3".Level;
      T     "Blend_T-30"."Dose_Level_%"."ChiliAwetan3%";


NETWORK
TITLE = Tomato to Blending T-30
//Valve Open
      A     "Preparation to Blend"."T-05_Tomato".Valve_Open;
      A(;
      O(;
      A     "Blend_T-30".Dose.Dose_Header_Req.%X3;
      A     "Blend_T-30".IN_FBAV_Header1;
      );
      O(;
      A     "Blend_T-30".Dose.Dose_Header_Req.%X19;
      A     "Blend_T-30".IN_FBAV_Header2;
      );
      );
      =     "Blend_T-30".Dose_Tomato.V_OPEN;
//Pump On
      O     "Preparation to Blend"."T-05_Tomato".Pump_Run;
      =     "Blend_T-30".Dose_Tomato.P_RUN;
//Tank Available
      O     "Preparation to Blend"."T-05_Tomato".Tank_Available;
      O     "Blend_T-30".Dose_Tomato.QDOSERun;
      =     "Blend_T-30".Dose.Dose_Tank_Available.%X3;
//Product Ready
      O     "Preparation to Blend"."T-05_Tomato".Product_Ready;
      =     "Blend_T-30".Dose.Dose_Prod_Ready.%X3;
//Level Tank
      L     "Preparation to Blend"."T-05_Tomato".Level;
      T     "Blend_T-30"."Dose_Level_%"."Tomato%";


NETWORK
TITLE = ChiliFresh1 to Blending T-30
//Valve Open
      A     "Preparation to Blend"."T-06_ChiliFresh_1".Valve_Open;
      A(;
      O(;
      A     "Blend_T-30".Dose.Dose_Header_Req.%X4;
      A     "Blend_T-30".IN_FBAV_Header1;
      );
      O(;
      A     "Blend_T-30".Dose.Dose_Header_Req.%X20;
      A     "Blend_T-30".IN_FBAV_Header2;
      );
      );
      =     "Blend_T-30".Dose_ChiliFresh1.V_OPEN;
//Pump On
      O     "Preparation to Blend"."T-06_ChiliFresh_1".Pump_Run;
      =     "Blend_T-30".Dose_ChiliFresh1.P_RUN;
//Tank Available
      O     "Preparation to Blend"."T-06_ChiliFresh_1".Tank_Available;
      O     "Blend_T-30".Dose_ChiliFresh1.QDOSERun;
      =     "Blend_T-30".Dose.Dose_Tank_Available.%X4;
//Product Ready
      O     "Preparation to Blend"."T-06_ChiliFresh_1".Product_Ready;
      =     "Blend_T-30".Dose.Dose_Prod_Ready.%X4;
//Level Tank
      L     "Preparation to Blend"."T-06_ChiliFresh_1".Level;
      T     "Blend_T-30"."Dose_Level_%"."ChiliFresh1%";


NETWORK
TITLE = ChiliFresh2 to Blending T-30
//Valve Open
      A     "Preparation to Blend"."T-07_ChiliFresh_2".Valve_Open;
      A(;
      O(;
      A     "Blend_T-30".Dose.Dose_Header_Req.%X5;
      A     "Blend_T-30".IN_FBAV_Header1;
      );
      O(;
      A     "Blend_T-30".Dose.Dose_Header_Req.%X21;
      A     "Blend_T-30".IN_FBAV_Header2;
      );
      );
      =     "Blend_T-30".Dose_ChiliFresh2.V_OPEN;
//Pump On
      O     "Preparation to Blend"."T-07_ChiliFresh_2".Pump_Run;
      =     "Blend_T-30".Dose_ChiliFresh2.P_RUN;
//Tank Available
      O     "Preparation to Blend"."T-07_ChiliFresh_2".Tank_Available;
      O     "Blend_T-30".Dose_ChiliFresh2.QDOSERun;
      =     "Blend_T-30".Dose.Dose_Tank_Available.%X5;
//Product Ready
      O     "Preparation to Blend"."T-07_ChiliFresh_2".Product_Ready;
      =     "Blend_T-30".Dose.Dose_Prod_Ready.%X5;
//Level Tank
      L     "Preparation to Blend"."T-07_ChiliFresh_2".Level;
      T     "Blend_T-30"."Dose_Level_%"."ChiliFresh2%";


NETWORK
TITLE = ChiliFresh3 to Blending T-30
//Valve Open
      A     "Preparation to Blend"."T-08_ChiliFresh_3".Valve_Open;
      A(;
      O(;
      A     "Blend_T-30".Dose.Dose_Header_Req.%X6;
      A     "Blend_T-30".IN_FBAV_Header1;
      );
      O(;
      A     "Blend_T-30".Dose.Dose_Header_Req.%X22;
      A     "Blend_T-30".IN_FBAV_Header2;
      );
      );
      =     "Blend_T-30".Dose_ChiliFresh3.V_OPEN;
//Pump On
      O     "Preparation to Blend"."T-08_ChiliFresh_3".Pump_Run;
      =     "Blend_T-30".Dose_ChiliFresh3.P_RUN;
//Tank Available
      O     "Preparation to Blend"."T-08_ChiliFresh_3".Tank_Available;
      O     "Blend_T-30".Dose_ChiliFresh3.QDOSERun;
      =     "Blend_T-30".Dose.Dose_Tank_Available.%X6;
//Product Ready
      O     "Preparation to Blend"."T-08_ChiliFresh_3".Product_Ready;
      =     "Blend_T-30".Dose.Dose_Prod_Ready.%X6;
//Level Tank
      L     "Preparation to Blend"."T-08_ChiliFresh_3".Level;
      T     "Blend_T-30"."Dose_Level_%"."ChiliFresh3%";


NETWORK
TITLE = Garlic to Blending T-30
//Valve Open
      A     "Preparation to Blend"."T-09_Garlic".Valve_Open;
      A(;
      O(;
      A     "Blend_T-30".Dose.Dose_Header_Req.%X7;
      A     "Blend_T-30".IN_FBAV_Header1;
      );
      O(;
      A     "Blend_T-30".Dose.Dose_Header_Req.%X23;
      A     "Blend_T-30".IN_FBAV_Header2;
      );
      );
      =     "Blend_T-30".Dose_Garlic.V_OPEN;
//Pump On
      O     "Preparation to Blend"."T-09_Garlic".Pump_Run;
      =     "Blend_T-30".Dose_Garlic.P_RUN;
//Tank Available
      O     "Preparation to Blend"."T-09_Garlic".Tank_Available;
      O     "Blend_T-30".Dose_Garlic.QDOSERun;
      =     "Blend_T-30".Dose.Dose_Tank_Available.%X7;
//Product Ready
      O     "Preparation to Blend"."T-09_Garlic".Product_Ready;
      =     "Blend_T-30".Dose.Dose_Prod_Ready.%X7;
//Level Tank
      L     "Preparation to Blend"."T-09_Garlic".Level;
      T     "Blend_T-30"."Dose_Level_%"."Garlic%";


NETWORK
TITLE = Vinegar to Blending T-30
//Valve Open
      A     "Preparation to Blend"."T-10_Vinegar".Valve_Open;
      A     "Blend_T-30".IN_FBAV_Vinegar;
      =     "Blend_T-30".Dose_Vinegar.V_OPEN;
//Pump On
      O     "Preparation to Blend"."T-10_Vinegar".Pump_Run;
      =     "Blend_T-30".Dose_Vinegar.P_RUN;
//Tank Available
      O     "Preparation to Blend"."T-10_Vinegar".Tank_Available;
      O     "Blend_T-30".Dose_Vinegar.QDOSERun;
      =     "Blend_T-30".Dose.Dose_Tank_Available.%X9;
//Product Ready
      O     "Preparation to Blend"."T-10_Vinegar".Product_Ready;
      =     "Blend_T-30".Dose.Dose_Prod_Ready.%X9;
//Level Tank
      L     "Preparation to Blend"."T-10_Vinegar".Level;
      T     "Blend_T-30"."Dose_Level_%"."Vinegar%";


NETWORK
TITLE = HW to Blending T-30
//Valve Open
      A     "Preparation to Blend"."T-51_HW".Valve_Open;
      A(;
      O(;
      A     "Blend_T-30".Dose.Dose_Header_Req.%X8;
      A     "Blend_T-30".IN_FBAV_Header1;
      );
      O(;
      A     "Blend_T-30".Dose.Dose_Header_Req.%X24;
      A     "Blend_T-30".IN_FBAV_Header2;
      );
      );
      =     "Blend_T-30".Dose_HW.V_OPEN;
//Pump On
      O     "Preparation to Blend"."T-51_HW".Pump_Run;
      =     "Blend_T-30".Dose_HW.P_RUN;
//Tank Available
      O     "Preparation to Blend"."T-51_HW".Tank_Available;
      O     "Blend_T-30".Dose_HW.QDOSERun;
      =     "Blend_T-30".Dose.Dose_Tank_Available.%X8;
//Product Ready
      O     "Preparation to Blend"."T-51_HW".Product_Ready;
      =     "Blend_T-30".Dose.Dose_Prod_Ready.%X8;
//Level Tank
// L     "Preparation to Blend"."T-01_HW".Level
// T     "Blend_T-30"."Dose_Level_%"."HW%"


REGION Network 55: Homomixer 13.00 to Blending T-30.00
   RUNG wire#powerrail
      Contact( "AlwaysTRUE" )
      wire#w1
      Contact( "IO Valve Homomixer_DB"."AV-13.03".FB_OPEN )
      Contact( "Blend_T-30".IN_FBAV_Homomixer )
      Coil( "Blend_T-30".Dose_Homomixer.V_OPEN )
   END_RUNG
   RUNG wire#w1
      Contact( "IO Valve Homomixer_DB"."P-13.01".FB_ON )
      Coil( "Blend_T-30".Dose_Homomixer.P_RUN )
   END_RUNG
   RUNG wire#w1
      Contact( "T-13.00_Homomixer".Out_Tank_Ready )
      wire#w2
      Coil( "Blend_T-30".Dose.Dose_Tank_Available.%X13 )
   END_RUNG
   RUNG wire#w1
      Contact( "Blend_T-30".Dose_Homomixer.QDOSERun )
   END_RUNG wire#w2
   RUNG wire#w1
      Contact( "T-13.00_Homomixer".Out_Prod_Ready )
      Coil( "Blend_T-30".Dose.Dose_Prod_Ready.%X13 )
   END_RUNG
   // the same network as SCL:
   "Blend_T-30".Dose_Homomixer.V_OPEN := "AlwaysTRUE" AND "IO Valve Homomixer_DB"."AV-13.03".FB_OPEN AND "Blend_T-30".IN_FBAV_Homomixer;
   "Blend_T-30".Dose_Homomixer.P_RUN := "AlwaysTRUE" AND "IO Valve Homomixer_DB"."P-13.01".FB_ON;
   "Blend_T-30".Dose.Dose_Tank_Available.%X13 := "AlwaysTRUE" AND ("T-13.00_Homomixer".Out_Tank_Ready OR "Blend_T-30".Dose_Homomixer.QDOSERun);
   "Blend_T-30".Dose.Dose_Prod_Ready.%X13 := "AlwaysTRUE" AND "T-13.00_Homomixer".Out_Prod_Ready;
END_REGION

